LIN {X -0.088,Y -552.932,Z 572.275,A 0.000,B 0.000,C 90.000,E1 265.527} C_DIS
LIN {X -0.264,Y -552.166,Z 572.267,A 0.000,B 0.000,C 90.000,E1 264.147} C_DIS
LIN {X 0.151,Y -551.255,Z 572.260,A 0.000,B 0.000,C 90.000,E1 262.704} C_DIS
LIN {X -0.031,Y -550.259,Z 572.253,A 0.000,B 0.000,C 90.000,E1 261.602} C_DIS
LIN {X -0.102,Y -548.526,Z 572.244,A 0.000,B 0.000,C 90.000,E1 259.926} C_DIS
LIN {X -0.023,Y -546.833,Z 572.235,A 0.000,B 0.000,C 90.000,E1 258.229} C_DIS
LIN {X 0.017,Y -545.061,Z 572.225,A 0.000,B 0.000,C 90.000,E1 256.533} C_DIS
LIN {X 0.274,Y -543.280,Z 572.216,A 0.000,B 0.000,C 90.000,E1 254.810} C_DIS
LIN {X -0.094,Y -541.576,Z 572.208,A 0.000,B 0.000,C 90.000,E1 253.433} C_DIS
LIN {X 0.029,Y -539.678,Z 572.200,A 0.000,B 0.000,C 90.000,E1 252.000} C_DIS
LIN {X 0.055,Y -538.028,Z 572.194,A 0.000,B 0.000,C 90.000,E1 250.859} C_DIS
LIN {X 0.231,Y -536.142,Z 572.187,A 0.000,B 0.000,C 90.000,E1 249.699} C_DIS
LIN {X 0.172,Y -534.661,Z 572.183,A 0.000,B 0.000,C 90.000,E1 248.847} C_DIS
LIN {X 0.198,Y -531.884,Z 572.175,A 0.000,B 0.000,C 90.000,E1 247.411} C_DIS
LIN {X -0.115,Y -528.234,Z 572.165,A 0.000,B 0.000,C 90.000,E1 245.717} C_DIS
LIN {X -0.200,Y -525.022,Z 572.157,A 0.000,B 0.000,C 90.000,E1 244.280} C_DIS
LIN {X 0.109,Y -521.645,Z 572.149,A 0.000,B 0.000,C 90.000,E1 242.794} C_DIS
LIN {X -0.018,Y -518.791,Z 572.143,A 0.000,B 0.000,C 90.000,E1 241.641} C_DIS
LIN {X 0.056,Y -515.801,Z 572.136,A 0.000,B 0.000,C 90.000,E1 240.461} C_DIS
LIN {X 0.080,Y -512.503,Z 572.129,A 0.000,B 0.000,C 90.000,E1 239.282} C_DIS
LIN {X 0.214,Y -508.339,Z 572.121,A 0.000,B 0.000,C 90.000,E1 237.788} C_DIS
LIN {X 0.164,Y -503.280,Z 572.111,A 0.000,B 0.000,C 90.000,E1 236.008} C_DIS
LIN {X -0.001,Y -499.031,Z 572.103,A 0.000,B 0.000,C 90.000,E1 234.529} C_DIS
LIN {X 0.032,Y -492.451,Z 572.090,A 0.000,B 0.000,C 90.000,E1 232.110} C_DIS
LIN {X -0.062,Y -486.845,Z 572.078,A 0.000,B 0.000,C 90.000,E1 229.989} C_DIS
LIN {X -0.046,Y -481.361,Z 572.066,A 0.000,B 0.000,C 90.000,E1 227.838} C_DIS
LIN {X 0.036,Y -476.717,Z 572.055,A 0.000,B 0.000,C 90.000,E1 225.972} C_DIS
LIN {X 0.030,Y -474.441,Z 572.050,A 0.000,B 0.000,C 90.000,E1 225.040} C_DIS
LIN {X 0.182,Y -470.757,Z 572.042,A 0.000,B 0.000,C 90.000,E1 223.461} C_DIS
LIN {X 0.020,Y -466.436,Z 572.031,A 0.000,B 0.000,C 90.000,E1 221.595} C_DIS
LIN {X -0.149,Y -461.582,Z 572.019,A 0.000,B 0.000,C 90.000,E1 219.402} C_DIS
LIN {X -0.024,Y -456.772,Z 572.006,A 0.000,B 0.000,C 90.000,E1 217.156} C_DIS
LIN {X 0.258,Y -453.476,Z 571.998,A 0.000,B 0.000,C 90.000,E1 215.518} C_DIS
LIN {X 0.076,Y -448.240,Z 571.983,A 0.000,B 0.000,C 90.000,E1 212.959} C_DIS
LIN {X 0.188,Y -443.956,Z 571.971,A 0.000,B 0.000,C 90.000,E1 210.669} C_DIS
LIN {X -0.141,Y -440.991,Z 571.961,A 0.000,B 0.000,C 90.000,E1 209.077} C_DIS
LIN {X 0.241,Y -438.187,Z 571.952,A 0.000,B 0.000,C 90.000,E1 207.385} C_DIS
LIN {X -0.204,Y -434.731,Z 571.941,A 0.000,B 0.000,C 90.000,E1 205.463} C_DIS
LIN {X 0.239,Y -432.507,Z 571.934,A 0.000,B 0.000,C 90.000,E1 204.079} C_DIS
LIN {X -0.109,Y -429.841,Z 571.925,A 0.000,B 0.000,C 90.000,E1 202.461} C_DIS
LIN {X -0.108,Y -426.345,Z 571.912,A 0.000,B 0.000,C 90.000,E1 200.120} C_DIS
LIN {X 0.253,Y -423.517,Z 571.901,A 0.000,B 0.000,C 90.000,E1 198.055} C_DIS
LIN {X 0.109,Y -419.981,Z 571.885,A 0.000,B 0.000,C 90.000,E1 195.371} C_DIS
LIN {X -0.104,Y -417.895,Z 571.876,A 0.000,B 0.000,C 90.000,E1 193.703} C_DIS
LIN {X 0.203,Y -415.958,Z 571.869,A 0.000,B 0.000,C 90.000,E1 192.299} C_DIS
LIN {X -0.089,Y -411.389,Z 571.849,A 0.000,B 0.000,C 90.000,E1 188.916} C_DIS
LIN {X 0.052,Y -408.670,Z 571.836,A 0.000,B 0.000,C 90.000,E1 186.486} C_DIS
LIN {X 0.014,Y -406.386,Z 571.825,A 0.000,B 0.000,C 90.000,E1 184.416} C_DIS
LIN {X 0.157,Y -402.836,Z 571.803,A 0.000,B 0.000,C 90.000,E1 180.573} C_DIS
LIN {X -0.095,Y -401.155,Z 571.790,A 0.000,B 0.000,C 90.000,E1 178.165} C_DIS
LIN {X 0.102,Y -400.219,Z 571.780,A 0.000,B 0.000,C 90.000,E1 176.388} C_DIS
LIN {X -0.205,Y -399.268,Z 571.764,A 0.000,B 0.000,C 90.000,E1 173.628} C_DIS
LIN {X 0.011,Y -398.849,Z 571.751,A 0.000,B 0.000,C 90.000,E1 171.141} C_DIS
LIN {X -0.098,Y -398.774,Z 571.739,A 0.000,B 0.000,C 90.000,E1 169.050} C_DIS
LIN {X -0.033,Y -399.127,Z 571.722,A 0.000,B 0.000,C 90.000,E1 165.880} C_DIS
LIN {X -0.088,Y -399.778,Z 571.708,A 0.000,B 0.000,C 90.000,E1 163.433} C_DIS
LIN {X 0.001,Y -400.656,Z 571.694,A 0.000,B 0.000,C 90.000,E1 160.967} C_DIS
LIN {X 0.142,Y -401.621,Z 571.683,A 0.000,B 0.000,C 90.000,E1 158.847} C_DIS
LIN {X -0.157,Y -402.652,Z 571.671,A 0.000,B 0.000,C 90.000,E1 156.794} C_DIS
LIN {X -0.149,Y -403.596,Z 571.661,A 0.000,B 0.000,C 90.000,E1 155.049} C_DIS
LIN {X 0.219,Y -404.546,Z 571.652,A 0.000,B 0.000,C 90.000,E1 153.256} C_DIS
LIN {X -0.108,Y -405.512,Z 571.642,A 0.000,B 0.000,C 90.000,E1 151.563} C_DIS
LIN {X 0.228,Y -406.196,Z 571.634,A 0.000,B 0.000,C 90.000,E1 150.127} C_DIS
LIN {X -0.131,Y -406.783,Z 571.627,A 0.000,B 0.000,C 90.000,E1 148.791} C_DIS
LIN {X -0.008,Y -407.394,Z 571.617,A 0.000,B 0.000,C 90.000,E1 147.041} C_DIS
LIN {X 0.005,Y -407.816,Z 571.607,A 0.000,B 0.000,C 90.000,E1 145.308} C_DIS
LIN {X 0.021,Y -408.164,Z 571.598,A 0.000,B 0.000,C 90.000,E1 143.577} C_DIS
LIN {X 0.198,Y -408.476,Z 571.588,A 0.000,B 0.000,C 90.000,E1 141.823} C_DIS
LIN {X -0.042,Y -408.720,Z 571.577,A 0.000,B 0.000,C 90.000,E1 139.784} C_DIS
LIN {X -0.059,Y -408.883,Z 571.569,A 0.000,B 0.000,C 90.000,E1 138.405} C_DIS
LIN {X 0.199,Y -408.999,Z 571.557,A 0.000,B 0.000,C 90.000,E1 136.296} C_DIS
LIN {X 0.018,Y -409.279,Z 571.544,A 0.000,B 0.000,C 90.000,E1 133.905} C_DIS
LIN {X 0.146,Y -409.500,Z 571.534,A 0.000,B 0.000,C 90.000,E1 132.162} C_DIS
LIN {X 0.148,Y -409.543,Z 571.527,A 0.000,B 0.000,C 90.000,E1 130.782} C_DIS
LIN {X -0.115,Y -409.440,Z 571.519,A 0.000,B 0.000,C 90.000,E1 129.439} C_DIS
LIN {X 0.232,Y -409.205,Z 571.512,A 0.000,B 0.000,C 90.000,E1 128.096} C_DIS
LIN {X 0.098,Y -415.513,Z 571.500,A 0.000,B 0.000,C 90.000,E1 125.964} C_DIS
LIN {X 0.182,Y -425.905,Z 571.477,A 0.000,B 0.000,C 90.000,E1 121.878} C_DIS
LIN {X 0.136,Y -430.920,Z 571.468,A 0.000,B 0.000,C 90.000,E1 120.207} C_DIS
LIN {X 0.004,Y -434.960,Z 571.458,A 0.000,B 0.000,C 90.000,E1 118.487} C_DIS
LIN {X -0.035,Y -434.992,Z 571.458,A 0.000,B 0.000,C 90.000,E1 118.487} C_DIS
LIN {X 0.108,Y -447.698,Z 571.455,A 0.000,B 0.000,C 90.000,E1 117.897} C_DIS
LIN {X -0.098,Y -466.481,Z 571.450,A 0.000,B 0.000,C 90.000,E1 117.052} C_DIS
LIN {X 0.200,Y -474.972,Z 571.448,A 0.000,B 0.000,C 90.000,E1 116.616} C_DIS
LIN {X 0.019,Y -488.662,Z 571.444,A 0.000,B 0.000,C 90.000,E1 115.976} C_DIS
LIN {X 0.304,Y -500.110,Z 571.441,A 0.000,B 0.000,C 90.000,E1 115.335} C_DIS
LIN {X 0.027,Y -511.511,Z 571.437,A 0.000,B 0.000,C 90.000,E1 114.719} C_DIS
LIN {X 0.078,Y -517.954,Z 571.435,A 0.000,B 0.000,C 90.000,E1 114.335} C_DIS
LIN {X -0.215,Y -527.586,Z 571.432,A 0.000,B 0.000,C 90.000,E1 113.770} C_DIS
LIN {X -0.042,Y -536.611,Z 571.429,A 0.000,B 0.000,C 90.000,E1 113.131} C_DIS
LIN {X 0.083,Y -540.758,Z 571.427,A 0.000,B 0.000,C 90.000,E1 112.823} C_DIS
LIN {X 0.012,Y -544.976,Z 571.425,A 0.000,B 0.000,C 90.000,E1 112.514} C_DIS
LIN {X 0.082,Y -550.454,Z 571.423,A 0.000,B 0.000,C 90.000,E1 112.078} C_DIS
LIN {X -0.089,Y -555.613,Z 571.420,A 0.000,B 0.000,C 90.000,E1 111.642} C_DIS
LIN {X 0.113,Y -560.392,Z 571.418,A 0.000,B 0.000,C 90.000,E1 111.173} C_DIS
LIN {X -0.204,Y -564.852,Z 571.415,A 0.000,B 0.000,C 90.000,E1 110.737} C_DIS
LIN {X 0.171,Y -570.133,Z 571.412,A 0.000,B 0.000,C 90.000,E1 110.066} C_DIS
LIN {X 0.048,Y -575.019,Z 571.408,A 0.000,B 0.000,C 90.000,E1 109.396} C_DIS
LIN {X -0.032,Y -579.407,Z 571.404,A 0.000,B 0.000,C 90.000,E1 108.725} C_DIS
LIN {X -0.160,Y -584.107,Z 571.400,A 0.000,B 0.000,C 90.000,E1 107.928} C_DIS
LIN {X 0.211,Y -587.650,Z 571.396,A 0.000,B 0.000,C 90.000,E1 107.221} C_DIS
LIN {X 0.061,Y -591.597,Z 571.391,A 0.000,B 0.000,C 90.000,E1 106.441} C_DIS
LIN {X -0.128,Y -595.301,Z 571.387,A 0.000,B 0.000,C 90.000,E1 105.662} C_DIS
LIN {X 0.290,Y -598.783,Z 571.383,A 0.000,B 0.000,C 90.000,E1 104.828} C_DIS
LIN {X -0.268,Y -603.045,Z 571.377,A 0.000,B 0.000,C 90.000,E1 103.828} C_DIS
LIN {X 0.148,Y -608.165,Z 571.369,A 0.000,B 0.000,C 90.000,E1 102.479} C_DIS
LIN {X -0.287,Y -612.155,Z 571.364,A 0.000,B 0.000,C 90.000,E1 101.478} C_DIS
LIN {X -0.079,Y -616.069,Z 571.358,A 0.000,B 0.000,C 90.000,E1 100.423} C_DIS
LIN {X 0.115,Y -621.760,Z 571.349,A 0.000,B 0.000,C 90.000,E1 98.859} C_DIS
LIN {X -0.188,Y -627.237,Z 571.341,A 0.000,B 0.000,C 90.000,E1 97.352} C_DIS
LIN {X -0.255,Y -631.446,Z 571.334,A 0.000,B 0.000,C 90.000,E1 96.087} C_DIS
LIN {X 0.295,Y -633.757,Z 571.330,A 0.000,B 0.000,C 90.000,E1 95.277} C_DIS
LIN {X -0.086,Y -636.518,Z 571.324,A 0.000,B 0.000,C 90.000,E1 94.302} C_DIS
LIN {X 0.210,Y -638.864,Z 571.318,A 0.000,B 0.000,C 90.000,E1 93.269} C_DIS
LIN {X -0.252,Y -639.970,Z 571.316,A 0.000,B 0.000,C 90.000,E1 92.808} C_DIS
LIN {X 0.301,Y -641.344,Z 571.311,A 0.000,B 0.000,C 90.000,E1 92.007} C_DIS
LIN {X 0.250,Y -642.504,Z 571.307,A 0.000,B 0.000,C 90.000,E1 91.260} C_DIS
LIN {X -0.038,Y -643.700,Z 571.302,A 0.000,B 0.000,C 90.000,E1 90.286} C_DIS
LIN {X -0.082,Y -644.228,Z 571.297,A 0.000,B 0.000,C 90.000,E1 89.542} C_DIS
LIN {X 0.105,Y -644.478,Z 571.295,A 0.000,B 0.000,C 90.000,E1 89.026} C_DIS
LIN {X -0.144,Y -644.538,Z 571.289,A 0.000,B 0.000,C 90.000,E1 88.051} C_DIS
LIN {X -0.184,Y -644.296,Z 571.285,A 0.000,B 0.000,C 90.000,E1 87.306} C_DIS
LIN {X 0.209,Y -643.628,Z 571.279,A 0.000,B 0.000,C 90.000,E1 86.274} C_DIS
LIN {X -0.051,Y -642.536,Z 571.274,A 0.000,B 0.000,C 90.000,E1 85.298} C_DIS
LIN {X -0.025,Y -641.619,Z 571.270,A 0.000,B 0.000,C 90.000,E1 84.546} C_DIS
LIN {X -0.318,Y -640.005,Z 571.264,A 0.000,B 0.000,C 90.000,E1 83.571} C_DIS
LIN {X 0.063,Y -638.030,Z 571.259,A 0.000,B 0.000,C 90.000,E1 82.534} C_DIS
LIN {X 0.058,Y -636.281,Z 571.254,A 0.000,B 0.000,C 90.000,E1 81.781} C_DIS
LIN {X 0.035,Y -634.447,Z 571.250,A 0.000,B 0.000,C 90.000,E1 81.027} C_DIS
LIN {X 0.236,Y -630.960,Z 571.243,A 0.000,B 0.000,C 90.000,E1 79.746} C_DIS
LIN {X -0.240,Y -627.112,Z 571.236,A 0.000,B 0.000,C 90.000,E1 78.522} C_DIS
LIN {X -0.028,Y -625.508,Z 571.233,A 0.000,B 0.000,C 90.000,E1 77.993} C_DIS
LIN {X -0.035,Y -622.884,Z 571.229,A 0.000,B 0.000,C 90.000,E1 77.229} C_DIS
LIN {X 0.148,Y -621.001,Z 571.226,A 0.000,B 0.000,C 90.000,E1 76.700} C_DIS
LIN {X 0.094,Y -617.927,Z 571.222,A 0.000,B 0.000,C 90.000,E1 75.936} C_DIS
LIN {X 0.005,Y -614.677,Z 571.218,A 0.000,B 0.000,C 90.000,E1 75.172} C_DIS
LIN {X -0.163,Y -610.597,Z 571.213,A 0.000,B 0.000,C 90.000,E1 74.283} C_DIS
LIN {X -0.214,Y -606.056,Z 571.208,A 0.000,B 0.000,C 90.000,E1 73.378} C_DIS
LIN {X 0.263,Y -601.137,Z 571.203,A 0.000,B 0.000,C 90.000,E1 72.417} C_DIS
LIN {X 0.212,Y -597.337,Z 571.199,A 0.000,B 0.000,C 90.000,E1 71.764} C_DIS
LIN {X 0.257,Y -592.101,Z 571.194,A 0.000,B 0.000,C 90.000,E1 70.967} C_DIS
LIN {X -0.176,Y -588.386,Z 571.191,A 0.000,B 0.000,C 90.000,E1 70.477} C_DIS
LIN {X -0.145,Y -583.261,Z 571.188,A 0.000,B 0.000,C 90.000,E1 69.806} C_DIS
LIN {X 0.068,Y -577.957,Z 571.184,A 0.000,B 0.000,C 90.000,E1 69.156} C_DIS
LIN {X -0.196,Y -573.030,Z 571.181,A 0.000,B 0.000,C 90.000,E1 68.646} C_DIS
LIN {X 0.178,Y -568.107,Z 571.179,A 0.000,B 0.000,C 90.000,E1 68.103} C_DIS
LIN {X -0.201,Y -563.053,Z 571.176,A 0.000,B 0.000,C 90.000,E1 67.667} C_DIS
LIN {X 0.152,Y -557.756,Z 571.173,A 0.000,B 0.000,C 90.000,E1 67.177} C_DIS
LIN {X -0.122,Y -553.146,Z 571.171,A 0.000,B 0.000,C 90.000,E1 66.847} C_DIS
LIN {X -0.080,Y -546.850,Z 571.169,A 0.000,B 0.000,C 90.000,E1 66.410} C_DIS
LIN {X 0.018,Y -542.062,Z 571.167,A 0.000,B 0.000,C 90.000,E1 66.102} C_DIS
LIN {X 0.139,Y -535.859,Z 571.165,A 0.000,B 0.000,C 90.000,E1 65.741} C_DIS
LIN {X 0.167,Y -527.281,Z 571.163,A 0.000,B 0.000,C 90.000,E1 65.305} C_DIS
LIN {X 0.065,Y -518.444,Z 571.161,A 0.000,B 0.000,C 90.000,E1 64.921} C_DIS
LIN {X -0.272,Y -511.248,Z 571.159,A 0.000,B 0.000,C 90.000,E1 64.665} C_DIS
LIN {X -0.146,Y -488.653,Z 571.154,A 0.000,B 0.000,C 90.000,E1 63.768} C_DIS
LIN {X 0.070,Y -473.164,Z 571.151,A 0.000,B 0.000,C 90.000,E1 63.127} C_DIS
LIN {X 0.116,Y -459.487,Z 571.148,A 0.000,B 0.000,C 90.000,E1 62.538} C_DIS
LIN {X -0.069,Y -456.318,Z 571.147,A 0.000,B 0.000,C 90.000,E1 62.410} C_DIS
LIN {X -0.110,Y -456.279,Z 571.147,A 0.000,B 0.000,C 90.000,E1 62.410} C_DIS
LIN {X 0.276,Y -455.533,Z 571.144,A 0.000,B 0.000,C 90.000,E1 61.897} C_DIS
LIN {X 0.040,Y -445.588,Z 571.119,A 0.000,B 0.000,C 90.000,E1 57.406} C_DIS
LIN {X 0.096,Y -443.812,Z 571.114,A 0.000,B 0.000,C 90.000,E1 56.421} C_DIS
LIN {X -0.115,Y -437.182,Z 571.098,A 0.000,B 0.000,C 90.000,E1 53.703} C_DIS
LIN {X -0.154,Y -437.181,Z 571.098,A 0.000,B 0.000,C 90.000,E1 53.703} C_DIS
LIN {X 0.077,Y -439.358,Z 571.088,A 0.000,B 0.000,C 90.000,E1 51.823} C_DIS
LIN {X 0.260,Y -441.594,Z 571.077,A 0.000,B 0.000,C 90.000,E1 49.828} C_DIS
LIN {X -0.151,Y -443.500,Z 571.068,A 0.000,B 0.000,C 90.000,E1 48.243} C_DIS
LIN {X 0.069,Y -445.310,Z 571.059,A 0.000,B 0.000,C 90.000,E1 46.581} C_DIS
LIN {X 0.013,Y -447.037,Z 571.050,A 0.000,B 0.000,C 90.000,E1 44.960} C_DIS
LIN {X -0.009,Y -448.128,Z 571.043,A 0.000,B 0.000,C 90.000,E1 43.662} C_DIS
LIN {X -0.023,Y -449.052,Z 571.035,A 0.000,B 0.000,C 90.000,E1 42.366} C_DIS
LIN {X 0.001,Y -449.622,Z 571.030,A 0.000,B 0.000,C 90.000,E1 41.391} C_DIS
LIN {X 0.034,Y -450.168,Z 571.023,A 0.000,B 0.000,C 90.000,E1 40.092} C_DIS
LIN {X 0.123,Y -450.506,Z 571.014,A 0.000,B 0.000,C 90.000,E1 38.463} C_DIS
LIN {X 0.176,Y -450.636,Z 571.010,A 0.000,B 0.000,C 90.000,E1 37.810} C_DIS
LIN {X -0.012,Y -450.526,Z 571.001,A 0.000,B 0.000,C 90.000,E1 36.217} C_DIS
LIN {X -0.103,Y -450.233,Z 570.992,A 0.000,B 0.000,C 90.000,E1 34.612} C_DIS
LIN {X -0.044,Y -449.765,Z 570.980,A 0.000,B 0.000,C 90.000,E1 32.339} C_DIS
LIN {X -0.092,Y -449.388,Z 570.967,A 0.000,B 0.000,C 90.000,E1 30.079} C_DIS
LIN {X 0.225,Y -449.212,Z 570.960,A 0.000,B 0.000,C 90.000,E1 28.743} C_DIS
LIN {X 0.179,Y -448.941,Z 570.951,A 0.000,B 0.000,C 90.000,E1 27.129} C_DIS
LIN {X -0.131,Y -448.623,Z 570.938,A 0.000,B 0.000,C 90.000,E1 24.899} C_DIS
LIN {X -0.107,Y -448.456,Z 570.927,A 0.000,B 0.000,C 90.000,E1 22.950} C_DIS
LIN {X -0.021,Y -448.482,Z 570.920,A 0.000,B 0.000,C 90.000,E1 21.642} C_DIS
LIN {X -0.210,Y -448.518,Z 570.908,A 0.000,B 0.000,C 90.000,E1 19.396} C_DIS
LIN {X 0.032,Y -448.730,Z 570.895,A 0.000,B 0.000,C 90.000,E1 17.094} C_DIS
LIN {X 0.008,Y -449.157,Z 570.882,A 0.000,B 0.000,C 90.000,E1 14.828} C_DIS
LIN {X 0.210,Y -449.882,Z 570.870,A 0.000,B 0.000,C 90.000,E1 12.535} C_DIS
LIN {X 0.144,Y -450.729,Z 570.859,A 0.000,B 0.000,C 90.000,E1 10.602} C_DIS
LIN {X 0.143,Y -451.978,Z 570.846,A 0.000,B 0.000,C 90.000,E1 8.341} C_DIS
LIN {X -0.128,Y -453.695,Z 570.832,A 0.000,B 0.000,C 90.000,E1 5.796} C_DIS
LIN {X -0.203,Y -455.559,Z 570.820,A 0.000,B 0.000,C 90.000,E1 3.555} C_DIS
LIN {X 0.012,Y -457.357,Z 570.809,A 0.000,B 0.000,C 90.000,E1 1.604} C_DIS
LIN {X 0.110,Y -460.029,Z 570.795,A 0.000,B 0.000,C 90.000,E1 359.141} C_DIS
LIN {X -0.066,Y -463.334,Z 570.781,A 0.000,B 0.000,C 90.000,E1 356.617} C_DIS
LIN {X -0.122,Y -466.013,Z 570.771,A 0.000,B 0.000,C 90.000,E1 354.723} C_DIS
LIN {X 0.246,Y -469.326,Z 570.758,A 0.000,B 0.000,C 90.000,E1 352.470} C_DIS
LIN {X -0.054,Y -472.137,Z 570.748,A 0.000,B 0.000,C 90.000,E1 350.622} C_DIS
LIN {X 0.155,Y -475.469,Z 570.736,A 0.000,B 0.000,C 90.000,E1 348.409} C_DIS
LIN {X 0.040,Y -479.382,Z 570.722,A 0.000,B 0.000,C 90.000,E1 345.936} C_DIS
LIN {X 0.012,Y -484.890,Z 570.705,A 0.000,B 0.000,C 90.000,E1 342.851} C_DIS
LIN {X -0.239,Y -488.408,Z 570.695,A 0.000,B 0.000,C 90.000,E1 341.040} C_DIS
LIN {X -0.282,Y -491.392,Z 570.686,A 0.000,B 0.000,C 90.000,E1 339.518} C_DIS
LIN {X -0.135,Y -493.688,Z 570.679,A 0.000,B 0.000,C 90.000,E1 338.284} C_DIS
LIN {X 0.100,Y -496.529,Z 570.671,A 0.000,B 0.000,C 90.000,E1 336.741} C_DIS
LIN {X 0.128,Y -499.231,Z 570.663,A 0.000,B 0.000,C 90.000,E1 335.229} C_DIS
LIN {X 0.044,Y -502.287,Z 570.652,A 0.000,B 0.000,C 90.000,E1 333.435} C_DIS
LIN {X -0.043,Y -504.697,Z 570.644,A 0.000,B 0.000,C 90.000,E1 331.948} C_DIS
LIN {X -0.091,Y -507.087,Z 570.636,A 0.000,B 0.000,C 90.000,E1 330.461} C_DIS
LIN {X 0.041,Y -510.039,Z 570.626,A 0.000,B 0.000,C 90.000,E1 328.663} C_DIS
LIN {X 0.141,Y -513.556,Z 570.614,A 0.000,B 0.000,C 90.000,E1 326.580} C_DIS
LIN {X 0.113,Y -516.619,Z 570.605,A 0.000,B 0.000,C 90.000,E1 324.815} C_DIS
LIN {X 0.222,Y -519.230,Z 570.596,A 0.000,B 0.000,C 90.000,E1 323.336} C_DIS
LIN {X 0.141,Y -523.486,Z 570.583,A 0.000,B 0.000,C 90.000,E1 321.009} C_DIS
LIN {X -0.202,Y -527.567,Z 570.572,A 0.000,B 0.000,C 90.000,E1 319.013} C_DIS
LIN {X -0.147,Y -532.109,Z 570.561,A 0.000,B 0.000,C 90.000,E1 316.986} C_DIS
LIN {X -0.308,Y -535.604,Z 570.553,A 0.000,B 0.000,C 90.000,E1 315.567} C_DIS
LIN {X 0.045,Y -536.440,Z 570.551,A 0.000,B 0.000,C 90.000,E1 315.243} C_DIS
LIN {X 0.001,Y -537.927,Z 570.548,A 0.000,B 0.000,C 90.000,E1 314.676} C_DIS
LIN {X -0.031,Y -539.815,Z 570.545,A 0.000,B 0.000,C 90.000,E1 314.109} C_DIS
LIN {X -0.240,Y -541.344,Z 570.543,A 0.000,B 0.000,C 90.000,E1 313.704} C_DIS
LIN {X 0.137,Y -542.937,Z 570.541,A 0.000,B 0.000,C 90.000,E1 313.380} C_DIS
LIN {X -0.045,Y -543.615,Z 570.540,A 0.000,B 0.000,C 90.000,E1 313.257} C_DIS
LIN {X 0.150,Y -544.524,Z 570.540,A 0.000,B 0.000,C 90.000,E1 313.095} C_DIS
LIN {X -0.056,Y -545.632,Z 570.539,A 0.000,B 0.000,C 90.000,E1 312.975} C_DIS
LIN {X -0.036,Y -547.549,Z 570.537,A 0.000,B 0.000,C 90.000,E1 312.690} C_DIS
LIN {X 0.125,Y -550.221,Z 570.535,A 0.000,B 0.000,C 90.000,E1 312.366} C_DIS
LIN {X -0.013,Y -551.276,Z 570.535,A 0.000,B 0.000,C 90.000,E1 312.243} C_DIS
LIN {X 0.208,Y -552.579,Z 570.534,A 0.000,B 0.000,C 90.000,E1 312.081} C_DIS
LIN {X -0.044,Y -560.700,Z 570.530,A 0.000,B 0.000,C 90.000,E1 311.391} C_DIS
LIN {X 0.050,Y -568.069,Z 570.527,A 0.000,B 0.000,C 90.000,E1 310.825} C_DIS
LIN {X -0.065,Y -578.642,Z 570.523,A 0.000,B 0.000,C 90.000,E1 310.092} C_DIS
LIN {X -0.148,Y -593.325,Z 570.517,A 0.000,B 0.000,C 90.000,E1 309.036} C_DIS
LIN {X -0.106,Y -598.899,Z 570.514,A 0.000,B 0.000,C 90.000,E1 308.588} C_DIS
LIN {X 0.204,Y -604.198,Z 570.512,A 0.000,B 0.000,C 90.000,E1 308.096} C_DIS
LIN {X 0.230,Y -611.884,Z 570.508,A 0.000,B 0.000,C 90.000,E1 307.363} C_DIS
LIN {X -0.178,Y -621.354,Z 570.502,A 0.000,B 0.000,C 90.000,E1 306.377} C_DIS
LIN {X -0.035,Y -626.861,Z 570.498,A 0.000,B 0.000,C 90.000,E1 305.724} C_DIS
LIN {X 0.145,Y -634.105,Z 570.494,A 0.000,B 0.000,C 90.000,E1 304.818} C_DIS
LIN {X 0.011,Y -638.081,Z 570.491,A 0.000,B 0.000,C 90.000,E1 304.326} C_DIS
LIN {X -0.058,Y -643.593,Z 570.487,A 0.000,B 0.000,C 90.000,E1 303.579} C_DIS
LIN {X -0.069,Y -648.508,Z 570.482,A 0.000,B 0.000,C 90.000,E1 302.832} C_DIS
LIN {X -0.116,Y -651.476,Z 570.480,A 0.000,B 0.000,C 90.000,E1 302.339} C_DIS
LIN {X 0.112,Y -654.579,Z 570.476,A 0.000,B 0.000,C 90.000,E1 301.720} C_DIS
LIN {X -0.143,Y -658.032,Z 570.472,A 0.000,B 0.000,C 90.000,E1 301.003} C_DIS
LIN {X -0.145,Y -660.216,Z 570.469,A 0.000,B 0.000,C 90.000,E1 300.512} C_DIS
LIN {X 0.232,Y -663.355,Z 570.465,A 0.000,B 0.000,C 90.000,E1 299.745} C_DIS
LIN {X 0.074,Y -666.218,Z 570.461,A 0.000,B 0.000,C 90.000,E1 299.027} C_DIS
LIN {X -0.055,Y -668.888,Z 570.457,A 0.000,B 0.000,C 90.000,E1 298.309} C_DIS
LIN {X -0.161,Y -671.387,Z 570.453,A 0.000,B 0.000,C 90.000,E1 297.590} C_DIS
LIN {X 0.007,Y -672.161,Z 570.452,A 0.000,B 0.000,C 90.000,E1 297.334} C_DIS
LIN {X 0.180,Y -673.103,Z 570.451,A 0.000,B 0.000,C 90.000,E1 297.078} C_DIS
LIN {X 0.110,Y -675.289,Z 570.447,A 0.000,B 0.000,C 90.000,E1 296.360} C_DIS
LIN {X 0.291,Y -675.857,Z 570.445,A 0.000,B 0.000,C 90.000,E1 296.104} C_DIS
LIN {X -0.240,Y -676.015,Z 570.443,A 0.000,B 0.000,C 90.000,E1 295.668} C_DIS
LIN {X -0.053,Y -675.810,Z 570.441,A 0.000,B 0.000,C 90.000,E1 295.412} C_DIS
LIN {X 0.133,Y -674.890,Z 570.440,A 0.000,B 0.000,C 90.000,E1 295.155} C_DIS
LIN {X 0.226,Y -674.324,Z 570.439,A 0.000,B 0.000,C 90.000,E1 295.027} C_DIS
LIN {X -0.204,Y -672.883,Z 570.438,A 0.000,B 0.000,C 90.000,E1 294.823} C_DIS
LIN {X -0.115,Y -671.963,Z 570.437,A 0.000,B 0.000,C 90.000,E1 294.695} C_DIS
LIN {X -0.308,Y -670.456,Z 570.437,A 0.000,B 0.000,C 90.000,E1 294.591} C_DIS
LIN {X -0.126,Y -669.413,Z 570.436,A 0.000,B 0.000,C 90.000,E1 294.515} C_DIS
LIN {X -0.016,Y -666.897,Z 570.435,A 0.000,B 0.000,C 90.000,E1 294.259} C_DIS
LIN {X 0.086,Y -665.372,Z 570.434,A 0.000,B 0.000,C 90.000,E1 294.131} C_DIS
LIN {X 0.061,Y -663.097,Z 570.434,A 0.000,B 0.000,C 90.000,E1 294.027} C_DIS
LIN {X 0.257,Y -657.087,Z 570.432,A 0.000,B 0.000,C 90.000,E1 293.770} C_DIS
LIN {X 0.090,Y -655.093,Z 570.432,A 0.000,B 0.000,C 90.000,E1 293.718} C_DIS
LIN {X -0.292,Y -646.617,Z 570.431,A 0.000,B 0.000,C 90.000,E1 293.515} C_DIS
LIN {X 0.153,Y -628.270,Z 570.428,A 0.000,B 0.000,C 90.000,E1 293.025} C_DIS
LIN {X -0.238,Y -621.422,Z 570.427,A 0.000,B 0.000,C 90.000,E1 292.898} C_DIS
LIN {X 0.179,Y -601.374,Z 570.424,A 0.000,B 0.000,C 90.000,E1 292.280} C_DIS
LIN {X -0.040,Y -580.842,Z 570.420,A 0.000,B 0.000,C 90.000,E1 291.642} C_DIS
LIN {X -0.054,Y -573.123,Z 570.419,A 0.000,B 0.000,C 90.000,E1 291.354} C_DIS
LIN {X -0.135,Y -567.535,Z 570.417,A 0.000,B 0.000,C 90.000,E1 291.099} C_DIS
LIN {X 0.028,Y -564.657,Z 570.416,A 0.000,B 0.000,C 90.000,E1 290.844} C_DIS
LIN {X -0.008,Y -564.624,Z 570.416,A 0.000,B 0.000,C 90.000,E1 290.844} C_DIS
LIN {X -0.016,Y -563.935,Z 570.415,A 0.000,B 0.000,C 90.000,E1 290.663} C_DIS
LIN {X 0.055,Y -563.651,Z 570.412,A 0.000,B 0.000,C 90.000,E1 290.174} C_DIS
LIN {X -0.099,Y -563.715,Z 570.406,A 0.000,B 0.000,C 90.000,E1 289.087} C_DIS
LIN {X -0.250,Y -563.588,Z 570.400,A 0.000,B 0.000,C 90.000,E1 288.000} C_DIS
LIN {X 0.134,Y -563.220,Z 570.394,A 0.000,B 0.000,C 90.000,E1 286.858} C_DIS
LIN {X 0.114,Y -562.582,Z 570.386,A 0.000,B 0.000,C 90.000,E1 285.481} C_DIS
LIN {X -0.071,Y -561.825,Z 570.378,A 0.000,B 0.000,C 90.000,E1 284.120} C_DIS
LIN {X -0.091,Y -560.706,Z 570.368,A 0.000,B 0.000,C 90.000,E1 282.187} C_DIS
LIN {X 0.118,Y -559.882,Z 570.360,A 0.000,B 0.000,C 90.000,E1 280.782} C_DIS
LIN {X -0.197,Y -558.918,Z 570.351,A 0.000,B 0.000,C 90.000,E1 279.151} C_DIS
LIN {X 0.203,Y -557.912,Z 570.338,A 0.000,B 0.000,C 90.000,E1 276.891} C_DIS
LIN {X 0.113,Y -557.375,Z 570.331,A 0.000,B 0.000,C 90.000,E1 275.511} C_DIS
LIN {X 0.136,Y -556.748,Z 570.321,A 0.000,B 0.000,C 90.000,E1 273.841} C_DIS
LIN {X 0.070,Y -556.230,Z 570.312,A 0.000,B 0.000,C 90.000,E1 272.178} C_DIS
LIN {X -0.080,Y -555.687,Z 570.304,A 0.000,B 0.000,C 90.000,E1 270.802} C_DIS
LIN {X 0.226,Y -555.222,Z 570.298,A 0.000,B 0.000,C 90.000,E1 269.656} C_DIS
LIN {X 0.131,Y -554.528,Z 570.289,A 0.000,B 0.000,C 90.000,E1 267.993} C_DIS
LIN {X -0.046,Y -553.898,Z 570.281,A 0.000,B 0.000,C 90.000,E1 266.617} C_DIS
LIN {X -0.140,Y -552.995,Z 570.272,A 0.000,B 0.000,C 90.000,E1 264.951} C_DIS
LIN {X 0.232,Y -552.180,Z 570.264,A 0.000,B 0.000,C 90.000,E1 263.514} C_DIS
LIN {X 0.058,Y -551.369,Z 570.258,A 0.000,B 0.000,C 90.000,E1 262.413} C_DIS
LIN {X -0.118,Y -550.350,Z 570.252,A 0.000,B 0.000,C 90.000,E1 261.310} C_DIS
LIN {X -0.186,Y -548.574,Z 570.242,A 0.000,B 0.000,C 90.000,E1 259.634} C_DIS
LIN {X -0.205,Y -547.174,Z 570.235,A 0.000,B 0.000,C 90.000,E1 258.229} C_DIS
LIN {X -0.029,Y -545.397,Z 570.225,A 0.000,B 0.000,C 90.000,E1 256.520} C_DIS
LIN {X 0.108,Y -543.583,Z 570.216,A 0.000,B 0.000,C 90.000,E1 254.810} C_DIS
LIN {X 0.266,Y -541.844,Z 570.208,A 0.000,B 0.000,C 90.000,E1 253.378} C_DIS
LIN {X -0.128,Y -539.912,Z 570.200,A 0.000,B 0.000,C 90.000,E1 252.000} C_DIS
LIN {X -0.097,Y -538.209,Z 570.194,A 0.000,B 0.000,C 90.000,E1 250.859} C_DIS
LIN {X -0.206,Y -535.813,Z 570.186,A 0.000,B 0.000,C 90.000,E1 249.444} C_DIS
LIN {X -0.265,Y -534.236,Z 570.181,A 0.000,B 0.000,C 90.000,E1 248.592} C_DIS
LIN {X 0.055,Y -532.011,Z 570.175,A 0.000,B 0.000,C 90.000,E1 247.411} C_DIS
LIN {X 0.227,Y -528.355,Z 570.165,A 0.000,B 0.000,C 90.000,E1 245.665} C_DIS
LIN {X 0.136,Y -525.115,Z 570.157,A 0.000,B 0.000,C 90.000,E1 244.229} C_DIS
LIN {X -0.025,Y -521.695,Z 570.149,A 0.000,B 0.000,C 90.000,E1 242.794} C_DIS
LIN {X -0.151,Y -518.826,Z 570.142,A 0.000,B 0.000,C 90.000,E1 241.641} C_DIS
LIN {X -0.077,Y -515.831,Z 570.136,A 0.000,B 0.000,C 90.000,E1 240.461} C_DIS
LIN {X -0.051,Y -512.531,Z 570.129,A 0.000,B 0.000,C 90.000,E1 239.282} C_DIS
LIN {X -0.012,Y -507.402,Z 570.120,A 0.000,B 0.000,C 90.000,E1 237.502} C_DIS
LIN {X 0.035,Y -503.184,Z 570.111,A 0.000,B 0.000,C 90.000,E1 236.008} C_DIS
LIN {X 0.276,Y -498.935,Z 570.103,A 0.000,B 0.000,C 90.000,E1 234.482} C_DIS
LIN {X -0.099,Y -492.378,Z 570.089,A 0.000,B 0.000,C 90.000,E1 232.110} C_DIS
LIN {X -0.193,Y -486.767,Z 570.078,A 0.000,B 0.000,C 90.000,E1 229.989} C_DIS
LIN {X 0.178,Y -481.295,Z 570.066,A 0.000,B 0.000,C 90.000,E1 227.796} C_DIS
LIN {X 0.126,Y -475.144,Z 570.052,A 0.000,B 0.000,C 90.000,E1 225.324} C_DIS
LIN {X 0.048,Y -470.689,Z 570.042,A 0.000,B 0.000,C 90.000,E1 223.461} C_DIS
LIN {X -0.184,Y -467.086,Z 570.033,A 0.000,B 0.000,C 90.000,E1 221.919} C_DIS
LIN {X -0.032,Y -462.151,Z 570.021,A 0.000,B 0.000,C 90.000,E1 219.688} C_DIS
LIN {X 0.244,Y -459.399,Z 570.013,A 0.000,B 0.000,C 90.000,E1 218.382} C_DIS
LIN {X -0.058,Y -455.325,Z 570.003,A 0.000,B 0.000,C 90.000,E1 216.503} C_DIS
LIN {X -0.157,Y -452.660,Z 569.996,A 0.000,B 0.000,C 90.000,E1 215.231} C_DIS
LIN {X -0.063,Y -448.112,Z 569.983,A 0.000,B 0.000,C 90.000,E1 212.959} C_DIS
LIN {X -0.017,Y -444.404,Z 569.972,A 0.000,B 0.000,C 90.000,E1 211.003} C_DIS
LIN {X 0.050,Y -441.451,Z 569.963,A 0.000,B 0.000,C 90.000,E1 209.361} C_DIS
LIN {X 0.095,Y -438.024,Z 569.952,A 0.000,B 0.000,C 90.000,E1 207.385} C_DIS
LIN {X 0.215,Y -435.164,Z 569.943,A 0.000,B 0.000,C 90.000,E1 205.720} C_DIS
LIN {X -0.101,Y -431.317,Z 569.930,A 0.000,B 0.000,C 90.000,E1 203.439} C_DIS
LIN {X -0.063,Y -426.718,Z 569.914,A 0.000,B 0.000,C 90.000,E1 200.429} C_DIS
LIN {X 0.120,Y -424.344,Z 569.904,A 0.000,B 0.000,C 90.000,E1 198.725} C_DIS
LIN {X -0.105,Y -421.587,Z 569.893,A 0.000,B 0.000,C 90.000,E1 196.732} C_DIS
LIN {X -0.229,Y -419.078,Z 569.882,A 0.000,B 0.000,C 90.000,E1 194.717} C_DIS
LIN {X 0.143,Y -417.823,Z 569.876,A 0.000,B 0.000,C 90.000,E1 193.647} C_DIS
LIN {X -0.007,Y -416.400,Z 569.870,A 0.000,B 0.000,C 90.000,E1 192.647} C_DIS
LIN {X 0.085,Y -412.186,Z 569.853,A 0.000,B 0.000,C 90.000,E1 189.557} C_DIS
LIN {X -0.106,Y -408.671,Z 569.836,A 0.000,B 0.000,C 90.000,E1 186.486} C_DIS
LIN {X -0.143,Y -406.412,Z 569.824,A 0.000,B 0.000,C 90.000,E1 184.416} C_DIS
LIN {X 0.003,Y -402.913,Z 569.803,A 0.000,B 0.000,C 90.000,E1 180.573} C_DIS
LIN {X 0.184,Y -401.471,Z 569.792,A 0.000,B 0.000,C 90.000,E1 178.453} C_DIS
LIN {X 0.000,Y -400.500,Z 569.782,A 0.000,B 0.000,C 90.000,E1 176.731} C_DIS
LIN {X 0.107,Y -399.470,Z 569.766,A 0.000,B 0.000,C 90.000,E1 173.913} C_DIS
LIN {X -0.132,Y -398.970,Z 569.751,A 0.000,B 0.000,C 90.000,E1 171.141} C_DIS
LIN {X 0.154,Y -398.895,Z 569.739,A 0.000,B 0.000,C 90.000,E1 168.993} C_DIS
LIN {X -0.168,Y -399.254,Z 569.721,A 0.000,B 0.000,C 90.000,E1 165.880} C_DIS
LIN {X 0.003,Y -399.711,Z 569.712,A 0.000,B 0.000,C 90.000,E1 164.102} C_DIS
LIN {X 0.165,Y -400.674,Z 569.696,A 0.000,B 0.000,C 90.000,E1 161.275} C_DIS
LIN {X -0.069,Y -401.620,Z 569.685,A 0.000,B 0.000,C 90.000,E1 159.209} C_DIS
LIN {X 0.006,Y -402.629,Z 569.673,A 0.000,B 0.000,C 90.000,E1 157.102} C_DIS
LIN {X 0.017,Y -403.595,Z 569.663,A 0.000,B 0.000,C 90.000,E1 155.357} C_DIS
LIN {X 0.104,Y -404.739,Z 569.652,A 0.000,B 0.000,C 90.000,E1 153.256} C_DIS
LIN {X 0.138,Y -405.720,Z 569.642,A 0.000,B 0.000,C 90.000,E1 151.513} C_DIS
LIN {X 0.120,Y -406.402,Z 569.634,A 0.000,B 0.000,C 90.000,E1 150.127} C_DIS
LIN {X 0.113,Y -407.008,Z 569.626,A 0.000,B 0.000,C 90.000,E1 148.742} C_DIS
LIN {X -0.109,Y -407.637,Z 569.617,A 0.000,B 0.000,C 90.000,E1 147.041} C_DIS
LIN {X -0.090,Y -408.057,Z 569.607,A 0.000,B 0.000,C 90.000,E1 145.308} C_DIS
LIN {X -0.070,Y -408.396,Z 569.598,A 0.000,B 0.000,C 90.000,E1 143.577} C_DIS
LIN {X 0.111,Y -408.698,Z 569.588,A 0.000,B 0.000,C 90.000,E1 141.823} C_DIS
LIN {X 0.149,Y -408.872,Z 569.580,A 0.000,B 0.000,C 90.000,E1 140.436} C_DIS
LIN {X -0.135,Y -409.069,Z 569.569,A 0.000,B 0.000,C 90.000,E1 138.405} C_DIS
LIN {X 0.127,Y -409.184,Z 569.557,A 0.000,B 0.000,C 90.000,E1 136.296} C_DIS
LIN {X 0.234,Y -409.462,Z 569.544,A 0.000,B 0.000,C 90.000,E1 133.866} C_DIS
LIN {X 0.082,Y -409.681,Z 569.534,A 0.000,B 0.000,C 90.000,E1 132.162} C_DIS
LIN {X 0.088,Y -409.724,Z 569.527,A 0.000,B 0.000,C 90.000,E1 130.782} C_DIS
LIN {X 0.087,Y -409.611,Z 569.519,A 0.000,B 0.000,C 90.000,E1 129.402} C_DIS
LIN {X -0.131,Y -409.346,Z 569.512,A 0.000,B 0.000,C 90.000,E1 128.096} C_DIS
LIN {X 0.043,Y -415.536,Z 569.500,A 0.000,B 0.000,C 90.000,E1 125.964} C_DIS
LIN {X 0.126,Y -425.926,Z 569.477,A 0.000,B 0.000,C 90.000,E1 121.878} C_DIS
LIN {X 0.080,Y -430.937,Z 569.468,A 0.000,B 0.000,C 90.000,E1 120.207} C_DIS
LIN {X -0.075,Y -435.623,Z 569.457,A 0.000,B 0.000,C 90.000,E1 118.231} C_DIS
LIN {X -0.112,Y -435.698,Z 569.457,A 0.000,B 0.000,C 90.000,E1 118.231} C_DIS
LIN {X -0.058,Y -442.880,Z 569.455,A 0.000,B 0.000,C 90.000,E1 117.897} C_DIS
LIN {X 0.248,Y -461.609,Z 569.450,A 0.000,B 0.000,C 90.000,E1 117.001} C_DIS
LIN {X 0.141,Y -470.241,Z 569.448,A 0.000,B 0.000,C 90.000,E1 116.616} C_DIS
LIN {X -0.246,Y -487.281,Z 569.443,A 0.000,B 0.000,C 90.000,E1 115.848} C_DIS
LIN {X 0.123,Y -498.819,Z 569.440,A 0.000,B 0.000,C 90.000,E1 115.207} C_DIS
LIN {X -0.066,Y -510.279,Z 569.437,A 0.000,B 0.000,C 90.000,E1 114.591} C_DIS
LIN {X 0.046,Y -516.743,Z 569.435,A 0.000,B 0.000,C 90.000,E1 114.207} C_DIS
LIN {X -0.150,Y -526.423,Z 569.431,A 0.000,B 0.000,C 90.000,E1 113.643} C_DIS
LIN {X 0.189,Y -537.119,Z 569.427,A 0.000,B 0.000,C 90.000,E1 112.898} C_DIS
LIN {X -0.065,Y -544.456,Z 569.424,A 0.000,B 0.000,C 90.000,E1 112.386} C_DIS
LIN {X 0.142,Y -549.034,Z 569.422,A 0.000,B 0.000,C 90.000,E1 112.025} C_DIS
LIN {X -0.032,Y -554.402,Z 569.420,A 0.000,B 0.000,C 90.000,E1 111.589} C_DIS
LIN {X 0.297,Y -559.475,Z 569.417,A 0.000,B 0.000,C 90.000,E1 111.099} C_DIS
LIN {X -0.029,Y -564.615,Z 569.415,A 0.000,B 0.000,C 90.000,E1 110.610} C_DIS
LIN {X -0.031,Y -569.267,Z 569.411,A 0.000,B 0.000,C 90.000,E1 110.066} C_DIS
LIN {X -0.161,Y -574.379,Z 569.408,A 0.000,B 0.000,C 90.000,E1 109.396} C_DIS
LIN {X 0.214,Y -579.703,Z 569.403,A 0.000,B 0.000,C 90.000,E1 108.544} C_DIS
LIN {X 0.171,Y -583.728,Z 569.399,A 0.000,B 0.000,C 90.000,E1 107.873} C_DIS
LIN {X -0.094,Y -588.065,Z 569.395,A 0.000,B 0.000,C 90.000,E1 107.094} C_DIS
LIN {X -0.245,Y -591.499,Z 569.391,A 0.000,B 0.000,C 90.000,E1 106.441} C_DIS
LIN {X 0.138,Y -595.322,Z 569.387,A 0.000,B 0.000,C 90.000,E1 105.607} C_DIS
LIN {X -0.016,Y -598.897,Z 569.382,A 0.000,B 0.000,C 90.000,E1 104.828} C_DIS
LIN {X 0.050,Y -605.410,Z 569.374,A 0.000,B 0.000,C 90.000,E1 103.244} C_DIS
LIN {X -0.080,Y -610.590,Z 569.366,A 0.000,B 0.000,C 90.000,E1 101.951} C_DIS
LIN {X -0.134,Y -615.559,Z 569.359,A 0.000,B 0.000,C 90.000,E1 100.658} C_DIS
LIN {X -0.179,Y -622.243,Z 569.349,A 0.000,B 0.000,C 90.000,E1 98.859} C_DIS
LIN {X -0.252,Y -626.844,Z 569.342,A 0.000,B 0.000,C 90.000,E1 97.587} C_DIS
LIN {X 0.256,Y -629.524,Z 569.338,A 0.000,B 0.000,C 90.000,E1 96.777} C_DIS
LIN {X -0.120,Y -632.849,Z 569.332,A 0.000,B 0.000,C 90.000,E1 95.796} C_DIS
LIN {X -0.248,Y -635.095,Z 569.328,A 0.000,B 0.000,C 90.000,E1 95.049} C_DIS
LIN {X 0.071,Y -637.791,Z 569.322,A 0.000,B 0.000,C 90.000,E1 94.012} C_DIS
LIN {X -0.260,Y -640.175,Z 569.317,A 0.000,B 0.000,C 90.000,E1 93.037} C_DIS
LIN {X 0.292,Y -641.626,Z 569.313,A 0.000,B 0.000,C 90.000,E1 92.236} C_DIS
LIN {X 0.244,Y -642.847,Z 569.308,A 0.000,B 0.000,C 90.000,E1 91.489} C_DIS
LIN {X 0.189,Y -643.843,Z 569.304,A 0.000,B 0.000,C 90.000,E1 90.745} C_DIS
LIN {X 0.146,Y -644.659,Z 569.300,A 0.000,B 0.000,C 90.000,E1 90.000} C_DIS
LIN {X -0.116,Y -645.176,Z 569.295,A 0.000,B 0.000,C 90.000,E1 89.026} C_DIS
LIN {X 0.289,Y -645.210,Z 569.289,A 0.000,B 0.000,C 90.000,E1 87.993} C_DIS
LIN {X 0.254,Y -644.952,Z 569.285,A 0.000,B 0.000,C 90.000,E1 87.249} C_DIS
LIN {X 0.014,Y -644.255,Z 569.279,A 0.000,B 0.000,C 90.000,E1 86.274} C_DIS
LIN {X -0.239,Y -643.124,Z 569.274,A 0.000,B 0.000,C 90.000,E1 85.298} C_DIS
LIN {X -0.206,Y -642.196,Z 569.270,A 0.000,B 0.000,C 90.000,E1 84.546} C_DIS
LIN {X 0.145,Y -640.522,Z 569.264,A 0.000,B 0.000,C 90.000,E1 83.514} C_DIS
LIN {X -0.103,Y -638.479,Z 569.259,A 0.000,B 0.000,C 90.000,E1 82.534} C_DIS
LIN {X -0.104,Y -636.723,Z 569.254,A 0.000,B 0.000,C 90.000,E1 81.781} C_DIS
LIN {X -0.120,Y -634.827,Z 569.250,A 0.000,B 0.000,C 90.000,E1 81.027} C_DIS
LIN {X 0.087,Y -631.268,Z 569.243,A 0.000,B 0.000,C 90.000,E1 79.746} C_DIS
LIN {X 0.232,Y -627.357,Z 569.236,A 0.000,B 0.000,C 90.000,E1 78.465} C_DIS
LIN {X -0.170,Y -625.719,Z 569.233,A 0.000,B 0.000,C 90.000,E1 77.993} C_DIS
LIN {X -0.174,Y -623.016,Z 569.229,A 0.000,B 0.000,C 90.000,E1 77.229} C_DIS
LIN {X 0.011,Y -621.091,Z 569.226,A 0.000,B 0.000,C 90.000,E1 76.700} C_DIS
LIN {X -0.042,Y -617.911,Z 569.222,A 0.000,B 0.000,C 90.000,E1 75.936} C_DIS
LIN {X -0.130,Y -614.565,Z 569.218,A 0.000,B 0.000,C 90.000,E1 75.172} C_DIS
LIN {X -0.094,Y -610.999,Z 569.213,A 0.000,B 0.000,C 90.000,E1 74.393} C_DIS
LIN {X -0.307,Y -606.381,Z 569.208,A 0.000,B 0.000,C 90.000,E1 73.504} C_DIS
LIN {X 0.171,Y -601.393,Z 569.203,A 0.000,B 0.000,C 90.000,E1 72.543} C_DIS
LIN {X 0.068,Y -596.649,Z 569.199,A 0.000,B 0.000,C 90.000,E1 71.764} C_DIS
LIN {X -0.180,Y -592.365,Z 569.195,A 0.000,B 0.000,C 90.000,E1 71.148} C_DIS
LIN {X -0.113,Y -587.581,Z 569.192,A 0.000,B 0.000,C 90.000,E1 70.477} C_DIS
LIN {X -0.090,Y -582.243,Z 569.188,A 0.000,B 0.000,C 90.000,E1 69.806} C_DIS
LIN {X -0.038,Y -577.612,Z 569.185,A 0.000,B 0.000,C 90.000,E1 69.263} C_DIS
LIN {X -0.006,Y -571.259,Z 569.181,A 0.000,B 0.000,C 90.000,E1 68.592} C_DIS
LIN {X -0.089,Y -567.335,Z 569.179,A 0.000,B 0.000,C 90.000,E1 68.209} C_DIS
LIN {X -0.254,Y -563.230,Z 569.177,A 0.000,B 0.000,C 90.000,E1 67.847} C_DIS
LIN {X -0.110,Y -557.511,Z 569.174,A 0.000,B 0.000,C 90.000,E1 67.358} C_DIS
LIN {X 0.138,Y -552.763,Z 569.172,A 0.000,B 0.000,C 90.000,E1 66.975} C_DIS
LIN {X 0.230,Y -546.382,Z 569.170,A 0.000,B 0.000,C 90.000,E1 66.538} C_DIS
LIN {X 0.052,Y -540.013,Z 569.168,A 0.000,B 0.000,C 90.000,E1 66.177} C_DIS
LIN {X -0.088,Y -533.449,Z 569.166,A 0.000,B 0.000,C 90.000,E1 65.845} C_DIS
LIN {X 0.141,Y -526.642,Z 569.164,A 0.000,B 0.000,C 90.000,E1 65.485} C_DIS
LIN {X -0.025,Y -516.116,Z 569.161,A 0.000,B 0.000,C 90.000,E1 65.049} C_DIS
LIN {X -0.284,Y -508.961,Z 569.160,A 0.000,B 0.000,C 90.000,E1 64.793} C_DIS
LIN {X -0.065,Y -486.236,Z 569.155,A 0.000,B 0.000,C 90.000,E1 63.896} C_DIS
LIN {X -0.072,Y -465.751,Z 569.150,A 0.000,B 0.000,C 90.000,E1 63.076} C_DIS
LIN {X 0.006,Y -456.823,Z 569.148,A 0.000,B 0.000,C 90.000,E1 62.666} C_DIS
LIN {X -0.033,Y -456.723,Z 569.148,A 0.000,B 0.000,C 90.000,E1 62.666} C_DIS
LIN {X 0.060,Y -455.612,Z 569.144,A 0.000,B 0.000,C 90.000,E1 61.975} C_DIS
LIN {X 0.147,Y -453.304,Z 569.139,A 0.000,B 0.000,C 90.000,E1 61.001} C_DIS
LIN {X -0.183,Y -444.503,Z 569.116,A 0.000,B 0.000,C 90.000,E1 56.834} C_DIS
LIN {X -0.122,Y -443.928,Z 569.114,A 0.000,B 0.000,C 90.000,E1 56.501} C_DIS
LIN {X 0.001,Y -437.569,Z 569.099,A 0.000,B 0.000,C 90.000,E1 53.863} C_DIS
LIN {X -0.038,Y -437.563,Z 569.099,A 0.000,B 0.000,C 90.000,E1 53.863} C_DIS
LIN {X -0.133,Y -439.942,Z 569.088,A 0.000,B 0.000,C 90.000,E1 51.904} C_DIS
LIN {X 0.101,Y -441.872,Z 569.079,A 0.000,B 0.000,C 90.000,E1 50.231} C_DIS
LIN {X -0.018,Y -443.836,Z 569.070,A 0.000,B 0.000,C 90.000,E1 48.609} C_DIS
LIN {X -0.106,Y -446.082,Z 569.059,A 0.000,B 0.000,C 90.000,E1 46.662} C_DIS
LIN {X 0.169,Y -447.821,Z 569.050,A 0.000,B 0.000,C 90.000,E1 45.000} C_DIS
LIN {X 0.156,Y -448.692,Z 569.045,A 0.000,B 0.000,C 90.000,E1 44.028} C_DIS
LIN {X -0.158,Y -449.642,Z 569.038,A 0.000,B 0.000,C 90.000,E1 42.771} C_DIS
LIN {X 0.175,Y -450.263,Z 569.032,A 0.000,B 0.000,C 90.000,E1 41.757} C_DIS
LIN {X 0.215,Y -450.833,Z 569.025,A 0.000,B 0.000,C 90.000,E1 40.458} C_DIS
LIN {X -0.024,Y -451.096,Z 569.020,A 0.000,B 0.000,C 90.000,E1 39.519} C_DIS
LIN {X 0.087,Y -451.363,Z 569.011,A 0.000,B 0.000,C 90.000,E1 37.890} C_DIS
LIN {X -0.083,Y -451.233,Z 569.002,A 0.000,B 0.000,C 90.000,E1 36.297} C_DIS
LIN {X 0.129,Y -450.999,Z 568.994,A 0.000,B 0.000,C 90.000,E1 34.978} C_DIS
LIN {X -0.160,Y -450.443,Z 568.982,A 0.000,B 0.000,C 90.000,E1 32.752} C_DIS
LIN {X 0.042,Y -450.028,Z 568.969,A 0.000,B 0.000,C 90.000,E1 30.463} C_DIS
LIN {X 0.148,Y -449.829,Z 568.962,A 0.000,B 0.000,C 90.000,E1 29.155} C_DIS
LIN {X -0.069,Y -449.539,Z 568.953,A 0.000,B 0.000,C 90.000,E1 27.564} C_DIS
LIN {X 0.034,Y -449.156,Z 568.941,A 0.000,B 0.000,C 90.000,E1 25.283} C_DIS
LIN {X -0.048,Y -448.892,Z 568.928,A 0.000,B 0.000,C 90.000,E1 23.025} C_DIS
LIN {X -0.071,Y -448.878,Z 568.919,A 0.000,B 0.000,C 90.000,E1 21.408} C_DIS
LIN {X 0.033,Y -448.863,Z 568.908,A 0.000,B 0.000,C 90.000,E1 19.450} C_DIS
LIN {X 0.147,Y -449.048,Z 568.896,A 0.000,B 0.000,C 90.000,E1 17.166} C_DIS
LIN {X 0.143,Y -449.431,Z 568.883,A 0.000,B 0.000,C 90.000,E1 14.898} C_DIS
LIN {X -0.018,Y -449.908,Z 568.874,A 0.000,B 0.000,C 90.000,E1 13.300} C_DIS
LIN {X -0.041,Y -450.934,Z 568.860,A 0.000,B 0.000,C 90.000,E1 10.715} C_DIS
LIN {X 0.159,Y -452.343,Z 568.845,A 0.000,B 0.000,C 90.000,E1 8.106} C_DIS
LIN {X 0.049,Y -454.331,Z 568.829,A 0.000,B 0.000,C 90.000,E1 5.220} C_DIS
LIN {X -0.012,Y -456.216,Z 568.817,A 0.000,B 0.000,C 90.000,E1 2.980} C_DIS
LIN {X -0.068,Y -458.387,Z 568.804,A 0.000,B 0.000,C 90.000,E1 0.745} C_DIS
LIN {X -0.209,Y -461.320,Z 568.790,A 0.000,B 0.000,C 90.000,E1 358.224} C_DIS
LIN {X -0.062,Y -463.459,Z 568.781,A 0.000,B 0.000,C 90.000,E1 356.617} C_DIS
LIN {X 0.144,Y -466.566,Z 568.769,A 0.000,B 0.000,C 90.000,E1 354.375} C_DIS
LIN {X 0.257,Y -469.420,Z 568.758,A 0.000,B 0.000,C 90.000,E1 352.470} C_DIS
LIN {X 0.211,Y -471.726,Z 568.750,A 0.000,B 0.000,C 90.000,E1 350.905} C_DIS
LIN {X -0.131,Y -475.036,Z 568.737,A 0.000,B 0.000,C 90.000,E1 348.757} C_DIS
LIN {X 0.096,Y -477.401,Z 568.729,A 0.000,B 0.000,C 90.000,E1 347.173} C_DIS
LIN {X -0.126,Y -480.447,Z 568.719,A 0.000,B 0.000,C 90.000,E1 345.338} C_DIS
LIN {X 0.031,Y -485.533,Z 568.703,A 0.000,B 0.000,C 90.000,E1 342.543} C_DIS
LIN {X -0.201,Y -489.059,Z 568.693,A 0.000,B 0.000,C 90.000,E1 340.732} C_DIS
LIN {X -0.228,Y -492.030,Z 568.684,A 0.000,B 0.000,C 90.000,E1 339.209} C_DIS
LIN {X -0.069,Y -494.265,Z 568.678,A 0.000,B 0.000,C 90.000,E1 337.975} C_DIS
LIN {X 0.174,Y -497.137,Z 568.669,A 0.000,B 0.000,C 90.000,E1 336.433} C_DIS
LIN {X -0.241,Y -499.825,Z 568.661,A 0.000,B 0.000,C 90.000,E1 334.973} C_DIS
LIN {X 0.137,Y -502.870,Z 568.651,A 0.000,B 0.000,C 90.000,E1 333.127} C_DIS
LIN {X 0.055,Y -505.263,Z 568.643,A 0.000,B 0.000,C 90.000,E1 331.641} C_DIS
LIN {X -0.062,Y -507.207,Z 568.636,A 0.000,B 0.000,C 90.000,E1 330.461} C_DIS
LIN {X -0.029,Y -510.654,Z 568.624,A 0.000,B 0.000,C 90.000,E1 328.377} C_DIS
LIN {X 0.094,Y -514.189,Z 568.613,A 0.000,B 0.000,C 90.000,E1 326.294} C_DIS
LIN {X 0.153,Y -516.765,Z 568.605,A 0.000,B 0.000,C 90.000,E1 324.815} C_DIS
LIN {X 0.263,Y -519.371,Z 568.596,A 0.000,B 0.000,C 90.000,E1 323.336} C_DIS
LIN {X 0.186,Y -523.618,Z 568.584,A 0.000,B 0.000,C 90.000,E1 321.009} C_DIS
LIN {X -0.152,Y -527.717,Z 568.572,A 0.000,B 0.000,C 90.000,E1 319.013} C_DIS
LIN {X 0.324,Y -531.574,Z 568.563,A 0.000,B 0.000,C 90.000,E1 317.229} C_DIS
LIN {X 0.037,Y -538.642,Z 568.547,A 0.000,B 0.000,C 90.000,E1 314.393} C_DIS
LIN {X -0.348,Y -540.565,Z 568.544,A 0.000,B 0.000,C 90.000,E1 313.866} C_DIS
LIN {X 0.024,Y -541.405,Z 568.542,A 0.000,B 0.000,C 90.000,E1 313.542} C_DIS
LIN {X 0.029,Y -542.433,Z 568.540,A 0.000,B 0.000,C 90.000,E1 313.257} C_DIS
LIN {X 0.012,Y -543.845,Z 568.539,A 0.000,B 0.000,C 90.000,E1 312.975} C_DIS
LIN {X 0.119,Y -545.997,Z 568.537,A 0.000,B 0.000,C 90.000,E1 312.609} C_DIS
LIN {X -0.034,Y -551.441,Z 568.533,A 0.000,B 0.000,C 90.000,E1 311.919} C_DIS
LIN {X 0.094,Y -555.851,Z 568.531,A 0.000,B 0.000,C 90.000,E1 311.472} C_DIS
LIN {X -0.012,Y -561.193,Z 568.528,A 0.000,B 0.000,C 90.000,E1 311.024} C_DIS
LIN {X -0.114,Y -569.835,Z 568.524,A 0.000,B 0.000,C 90.000,E1 310.378} C_DIS
LIN {X -0.140,Y -577.457,Z 568.521,A 0.000,B 0.000,C 90.000,E1 309.850} C_DIS
LIN {X 0.200,Y -592.164,Z 568.515,A 0.000,B 0.000,C 90.000,E1 308.749} C_DIS
LIN {X -0.100,Y -597.656,Z 568.513,A 0.000,B 0.000,C 90.000,E1 308.338} C_DIS
LIN {X -0.271,Y -603.006,Z 568.510,A 0.000,B 0.000,C 90.000,E1 307.890} C_DIS
LIN {X -0.285,Y -610.705,Z 568.506,A 0.000,B 0.000,C 90.000,E1 307.156} C_DIS
LIN {X -0.038,Y -616.678,Z 568.503,A 0.000,B 0.000,C 90.000,E1 306.503} C_DIS
LIN {X 0.264,Y -620.191,Z 568.501,A 0.000,B 0.000,C 90.000,E1 306.091} C_DIS
LIN {X 0.118,Y -625.601,Z 568.497,A 0.000,B 0.000,C 90.000,E1 305.471} C_DIS
LIN {X -0.230,Y -631.976,Z 568.493,A 0.000,B 0.000,C 90.000,E1 304.739} C_DIS
LIN {X 0.153,Y -636.986,Z 568.489,A 0.000,B 0.000,C 90.000,E1 304.072} C_DIS
LIN {X -0.082,Y -643.482,Z 568.485,A 0.000,B 0.000,C 90.000,E1 303.214} C_DIS
LIN {X 0.031,Y -646.797,Z 568.482,A 0.000,B 0.000,C 90.000,E1 302.704} C_DIS
LIN {X 0.013,Y -650.475,Z 568.478,A 0.000,B 0.000,C 90.000,E1 302.084} C_DIS
LIN {X -0.112,Y -651.731,Z 568.477,A 0.000,B 0.000,C 90.000,E1 301.848} C_DIS
LIN {X 0.193,Y -653.071,Z 568.476,A 0.000,B 0.000,C 90.000,E1 301.592} C_DIS
LIN {X -0.075,Y -656.502,Z 568.472,A 0.000,B 0.000,C 90.000,E1 300.875} C_DIS
LIN {X 0.151,Y -660.789,Z 568.466,A 0.000,B 0.000,C 90.000,E1 299.873} C_DIS
LIN {X -0.033,Y -663.735,Z 568.462,A 0.000,B 0.000,C 90.000,E1 299.155} C_DIS
LIN {X -0.037,Y -667.311,Z 568.457,A 0.000,B 0.000,C 90.000,E1 298.180} C_DIS
LIN {X 0.172,Y -671.552,Z 568.450,A 0.000,B 0.000,C 90.000,E1 296.950} C_DIS
LIN {X -0.088,Y -673.026,Z 568.447,A 0.000,B 0.000,C 90.000,E1 296.488} C_DIS
LIN {X 0.087,Y -673.636,Z 568.446,A 0.000,B 0.000,C 90.000,E1 296.232} C_DIS
LIN {X -0.166,Y -674.302,Z 568.443,A 0.000,B 0.000,C 90.000,E1 295.771} C_DIS
LIN {X -0.278,Y -674.219,Z 568.442,A 0.000,B 0.000,C 90.000,E1 295.540} C_DIS
LIN {X 0.083,Y -672.415,Z 568.439,A 0.000,B 0.000,C 90.000,E1 295.027} C_DIS
LIN {X 0.258,Y -671.004,Z 568.438,A 0.000,B 0.000,C 90.000,E1 294.771} C_DIS
LIN {X 0.172,Y -665.772,Z 568.435,A 0.000,B 0.000,C 90.000,E1 294.259} C_DIS
LIN {X 0.002,Y -663.968,Z 568.434,A 0.000,B 0.000,C 90.000,E1 294.155} C_DIS
LIN {X 0.120,Y -659.146,Z 568.433,A 0.000,B 0.000,C 90.000,E1 293.951} C_DIS
LIN {X 0.069,Y -656.575,Z 568.432,A 0.000,B 0.000,C 90.000,E1 293.823} C_DIS
LIN {X -0.154,Y -654.584,Z 568.432,A 0.000,B 0.000,C 90.000,E1 293.770} C_DIS
LIN {X -0.113,Y -651.959,Z 568.432,A 0.000,B 0.000,C 90.000,E1 293.695} C_DIS
LIN {X -0.016,Y -649.002,Z 568.431,A 0.000,B 0.000,C 90.000,E1 293.590} C_DIS
LIN {X -0.322,Y -645.435,Z 568.431,A 0.000,B 0.000,C 90.000,E1 293.515} C_DIS
LIN {X -0.158,Y -633.935,Z 568.429,A 0.000,B 0.000,C 90.000,E1 293.206} C_DIS
LIN {X 0.323,Y -620.392,Z 568.427,A 0.000,B 0.000,C 90.000,E1 292.823} C_DIS
LIN {X -0.201,Y -599.910,Z 568.424,A 0.000,B 0.000,C 90.000,E1 292.280} C_DIS
LIN {X 0.015,Y -579.360,Z 568.420,A 0.000,B 0.000,C 90.000,E1 291.589} C_DIS
LIN {X 0.054,Y -573.357,Z 568.419,A 0.000,B 0.000,C 90.000,E1 291.354} C_DIS
LIN {X 0.071,Y -568.226,Z 568.417,A 0.000,B 0.000,C 90.000,E1 291.099} C_DIS
LIN {X -0.211,Y -566.974,Z 568.417,A 0.000,B 0.000,C 90.000,E1 291.046} C_DIS
LIN {X 0.024,Y -565.161,Z 568.416,A 0.000,B 0.000,C 90.000,E1 290.865} C_DIS
LIN {X -0.013,Y -565.144,Z 568.416,A 0.000,B 0.000,C 90.000,E1 290.865} C_DIS
LIN {X 0.176,Y -564.529,Z 568.415,A 0.000,B 0.000,C 90.000,E1 290.684} C_DIS
LIN {X 0.077,Y -564.341,Z 568.414,A 0.000,B 0.000,C 90.000,E1 290.556} C_DIS
LIN {X 0.303,Y -564.155,Z 568.412,A 0.000,B 0.000,C 90.000,E1 290.120} C_DIS
LIN {X 0.159,Y -564.189,Z 568.406,A 0.000,B 0.000,C 90.000,E1 289.033} C_DIS
LIN {X 0.018,Y -564.078,Z 568.400,A 0.000,B 0.000,C 90.000,E1 287.946} C_DIS
LIN {X -0.128,Y -563.705,Z 568.394,A 0.000,B 0.000,C 90.000,E1 286.858} C_DIS
LIN {X -0.138,Y -563.061,Z 568.386,A 0.000,B 0.000,C 90.000,E1 285.481} C_DIS
LIN {X 0.231,Y -562.307,Z 568.378,A 0.000,B 0.000,C 90.000,E1 284.064} C_DIS
LIN {X -0.205,Y -561.192,Z 568.368,A 0.000,B 0.000,C 90.000,E1 282.175} C_DIS
LIN {X 0.047,Y -560.186,Z 568.358,A 0.000,B 0.000,C 90.000,E1 280.489} C_DIS
LIN {X 0.143,Y -559.393,Z 568.351,A 0.000,B 0.000,C 90.000,E1 279.095} C_DIS
LIN {X -0.195,Y -558.670,Z 568.341,A 0.000,B 0.000,C 90.000,E1 277.466} C_DIS
LIN {X -0.147,Y -557.977,Z 568.332,A 0.000,B 0.000,C 90.000,E1 275.796} C_DIS
LIN {X -0.041,Y -557.234,Z 568.321,A 0.000,B 0.000,C 90.000,E1 273.841} C_DIS
LIN {X -0.095,Y -556.696,Z 568.312,A 0.000,B 0.000,C 90.000,E1 272.178} C_DIS
LIN {X -0.238,Y -556.135,Z 568.304,A 0.000,B 0.000,C 90.000,E1 270.802} C_DIS
LIN {X 0.075,Y -555.667,Z 568.298,A 0.000,B 0.000,C 90.000,E1 269.656} C_DIS
LIN {X -0.011,Y -554.961,Z 568.289,A 0.000,B 0.000,C 90.000,E1 267.993} C_DIS
LIN {X -0.181,Y -554.294,Z 568.281,A 0.000,B 0.000,C 90.000,E1 266.617} C_DIS
LIN {X -0.266,Y -553.388,Z 568.272,A 0.000,B 0.000,C 90.000,E1 264.951} C_DIS
LIN {X 0.113,Y -552.555,Z 568.264,A 0.000,B 0.000,C 90.000,E1 263.514} C_DIS
LIN {X -0.055,Y -551.754,Z 568.258,A 0.000,B 0.000,C 90.000,E1 262.413} C_DIS
LIN {X -0.225,Y -550.747,Z 568.252,A 0.000,B 0.000,C 90.000,E1 261.310} C_DIS
LIN {X 0.245,Y -549.250,Z 568.244,A 0.000,B 0.000,C 90.000,E1 259.859} C_DIS
LIN {X 0.240,Y -547.522,Z 568.234,A 0.000,B 0.000,C 90.000,E1 258.173} C_DIS
LIN {X -0.114,Y -545.754,Z 568.225,A 0.000,B 0.000,C 90.000,E1 256.520} C_DIS
LIN {X 0.032,Y -543.895,Z 568.216,A 0.000,B 0.000,C 90.000,E1 254.810} C_DIS
LIN {X 0.195,Y -542.126,Z 568.208,A 0.000,B 0.000,C 90.000,E1 253.378} C_DIS
LIN {X -0.192,Y -540.157,Z 568.200,A 0.000,B 0.000,C 90.000,E1 252.000} C_DIS
LIN {X 0.061,Y -537.945,Z 568.192,A 0.000,B 0.000,C 90.000,E1 250.550} C_DIS
LIN {X -0.050,Y -535.516,Z 568.184,A 0.000,B 0.000,C 90.000,E1 249.135} C_DIS
LIN {X -0.199,Y -532.711,Z 568.176,A 0.000,B 0.000,C 90.000,E1 247.720} C_DIS
LIN {X 0.101,Y -530.313,Z 568.170,A 0.000,B 0.000,C 90.000,E1 246.538} C_DIS
LIN {X -0.122,Y -527.831,Z 568.163,A 0.000,B 0.000,C 90.000,E1 245.409} C_DIS
LIN {X 0.009,Y -524.541,Z 568.155,A 0.000,B 0.000,C 90.000,E1 243.948} C_DIS
LIN {X 0.074,Y -521.066,Z 568.147,A 0.000,B 0.000,C 90.000,E1 242.487} C_DIS
LIN {X 0.180,Y -518.135,Z 568.141,A 0.000,B 0.000,C 90.000,E1 241.307} C_DIS
LIN {X -0.119,Y -515.890,Z 568.136,A 0.000,B 0.000,C 90.000,E1 240.461} C_DIS
LIN {X 0.258,Y -513.446,Z 568.131,A 0.000,B 0.000,C 90.000,E1 239.537} C_DIS
LIN {X -0.054,Y -507.369,Z 568.119,A 0.000,B 0.000,C 90.000,E1 237.502} C_DIS
LIN {X -0.006,Y -503.116,Z 568.111,A 0.000,B 0.000,C 90.000,E1 236.008} C_DIS
LIN {X 0.234,Y -498.866,Z 568.103,A 0.000,B 0.000,C 90.000,E1 234.482} C_DIS
LIN {X 0.001,Y -493.125,Z 568.091,A 0.000,B 0.000,C 90.000,E1 232.396} C_DIS
LIN {X 0.099,Y -489.848,Z 568.084,A 0.000,B 0.000,C 90.000,E1 231.170} C_DIS
LIN {X -0.093,Y -485.920,Z 568.076,A 0.000,B 0.000,C 90.000,E1 229.666} C_DIS
LIN {X 0.133,Y -481.254,Z 568.066,A 0.000,B 0.000,C 90.000,E1 227.796} C_DIS
LIN {X 0.079,Y -475.070,Z 568.052,A 0.000,B 0.000,C 90.000,E1 225.324} C_DIS
LIN {X 0.001,Y -470.643,Z 568.042,A 0.000,B 0.000,C 90.000,E1 223.461} C_DIS
LIN {X -0.231,Y -467.028,Z 568.033,A 0.000,B 0.000,C 90.000,E1 221.919} C_DIS
LIN {X -0.126,Y -462.746,Z 568.022,A 0.000,B 0.000,C 90.000,E1 220.011} C_DIS
LIN {X -0.194,Y -460.042,Z 568.015,A 0.000,B 0.000,C 90.000,E1 218.749} C_DIS
LIN {X 0.160,Y -455.901,Z 568.005,A 0.000,B 0.000,C 90.000,E1 216.790} C_DIS
LIN {X -0.210,Y -452.556,Z 567.996,A 0.000,B 0.000,C 90.000,E1 215.231} C_DIS
LIN {X -0.196,Y -448.660,Z 567.985,A 0.000,B 0.000,C 90.000,E1 213.293} C_DIS
LIN {X -0.138,Y -444.879,Z 567.974,A 0.000,B 0.000,C 90.000,E1 211.337} C_DIS
LIN {X 0.158,Y -441.917,Z 567.965,A 0.000,B 0.000,C 90.000,E1 209.667} C_DIS
LIN {X 0.034,Y -437.890,Z 567.952,A 0.000,B 0.000,C 90.000,E1 207.385} C_DIS
LIN {X -0.024,Y -434.485,Z 567.941,A 0.000,B 0.000,C 90.000,E1 205.412} C_DIS
LIN {X 0.045,Y -430.651,Z 567.928,A 0.000,B 0.000,C 90.000,E1 203.078} C_DIS
LIN {X -0.133,Y -426.603,Z 567.913,A 0.000,B 0.000,C 90.000,E1 200.429} C_DIS
LIN {X -0.144,Y -424.725,Z 567.906,A 0.000,B 0.000,C 90.000,E1 199.087} C_DIS
LIN {X 0.046,Y -421.971,Z 567.895,A 0.000,B 0.000,C 90.000,E1 197.040} C_DIS
LIN {X 0.045,Y -419.442,Z 567.883,A 0.000,B 0.000,C 90.000,E1 195.009} C_DIS
LIN {X 0.069,Y -417.778,Z 567.876,A 0.000,B 0.000,C 90.000,E1 193.647} C_DIS
LIN {X -0.081,Y -416.341,Z 567.870,A 0.000,B 0.000,C 90.000,E1 192.647} C_DIS
LIN {X -0.031,Y -412.592,Z 567.855,A 0.000,B 0.000,C 90.000,E1 189.905} C_DIS
LIN {X 0.179,Y -410.118,Z 567.844,A 0.000,B 0.000,C 90.000,E1 187.814} C_DIS
LIN {X -0.207,Y -408.293,Z 567.834,A 0.000,B 0.000,C 90.000,E1 186.144} C_DIS
LIN {X 0.187,Y -406.460,Z 567.824,A 0.000,B 0.000,C 90.000,E1 184.359} C_DIS
LIN {X -0.068,Y -402.999,Z 567.803,A 0.000,B 0.000,C 90.000,E1 180.573} C_DIS
LIN {X 0.115,Y -401.558,Z 567.792,A 0.000,B 0.000,C 90.000,E1 178.453} C_DIS
LIN {X -0.067,Y -400.587,Z 567.782,A 0.000,B 0.000,C 90.000,E1 176.731} C_DIS
LIN {X 0.043,Y -399.559,Z 567.766,A 0.000,B 0.000,C 90.000,E1 173.913} C_DIS
LIN {X -0.175,Y -399.137,Z 567.753,A 0.000,B 0.000,C 90.000,E1 171.489} C_DIS
LIN {X 0.097,Y -399.019,Z 567.739,A 0.000,B 0.000,C 90.000,E1 168.993} C_DIS
LIN {X -0.222,Y -399.378,Z 567.721,A 0.000,B 0.000,C 90.000,E1 165.880} C_DIS
LIN {X -0.019,Y -399.764,Z 567.714,A 0.000,B 0.000,C 90.000,E1 164.448} C_DIS
LIN {X 0.033,Y -400.653,Z 567.698,A 0.000,B 0.000,C 90.000,E1 161.638} C_DIS
LIN {X 0.176,Y -401.606,Z 567.686,A 0.000,B 0.000,C 90.000,E1 159.518} C_DIS
LIN {X 0.097,Y -402.616,Z 567.675,A 0.000,B 0.000,C 90.000,E1 157.433} C_DIS
LIN {X -0.019,Y -403.773,Z 567.663,A 0.000,B 0.000,C 90.000,E1 155.357} C_DIS
LIN {X 0.072,Y -404.924,Z 567.652,A 0.000,B 0.000,C 90.000,E1 153.256} C_DIS
LIN {X 0.110,Y -405.921,Z 567.642,A 0.000,B 0.000,C 90.000,E1 151.513} C_DIS
LIN {X 0.095,Y -406.609,Z 567.634,A 0.000,B 0.000,C 90.000,E1 150.127} C_DIS
LIN {X 0.091,Y -407.228,Z 567.626,A 0.000,B 0.000,C 90.000,E1 148.742} C_DIS
LIN {X -0.126,Y -407.869,Z 567.617,A 0.000,B 0.000,C 90.000,E1 147.041} C_DIS
LIN {X -0.103,Y -408.295,Z 567.607,A 0.000,B 0.000,C 90.000,E1 145.308} C_DIS
LIN {X -0.077,Y -408.637,Z 567.598,A 0.000,B 0.000,C 90.000,E1 143.577} C_DIS
LIN {X 0.109,Y -408.933,Z 567.588,A 0.000,B 0.000,C 90.000,E1 141.823} C_DIS
LIN {X 0.151,Y -409.094,Z 567.580,A 0.000,B 0.000,C 90.000,E1 140.436} C_DIS
LIN {X 0.027,Y -409.249,Z 567.571,A 0.000,B 0.000,C 90.000,E1 138.728} C_DIS
LIN {X -0.009,Y -409.338,Z 567.559,A 0.000,B 0.000,C 90.000,E1 136.662} C_DIS
LIN {X -0.180,Y -409.588,Z 567.546,A 0.000,B 0.000,C 90.000,E1 134.271} C_DIS
LIN {X -0.050,Y -409.837,Z 567.536,A 0.000,B 0.000,C 90.000,E1 132.528} C_DIS
LIN {X -0.045,Y -409.932,Z 567.529,A 0.000,B 0.000,C 90.000,E1 131.148} C_DIS
LIN {X -0.044,Y -409.837,Z 567.521,A 0.000,B 0.000,C 90.000,E1 129.769} C_DIS
LIN {X -0.149,Y -409.694,Z 567.515,A 0.000,B 0.000,C 90.000,E1 128.749} C_DIS
LIN {X -0.143,Y -409.574,Z 567.511,A 0.000,B 0.000,C 90.000,E1 128.016} C_DIS
LIN {X 0.075,Y -415.522,Z 567.500,A 0.000,B 0.000,C 90.000,E1 125.964} C_DIS
LIN {X 0.159,Y -425.914,Z 567.477,A 0.000,B 0.000,C 90.000,E1 121.878} C_DIS
LIN {X 0.113,Y -430.927,Z 567.468,A 0.000,B 0.000,C 90.000,E1 120.207} C_DIS
LIN {X -0.141,Y -436.293,Z 567.455,A 0.000,B 0.000,C 90.000,E1 117.975} C_DIS
LIN {X -0.181,Y -436.358,Z 567.455,A 0.000,B 0.000,C 90.000,E1 117.975} C_DIS
LIN {X -0.052,Y -444.381,Z 567.453,A 0.000,B 0.000,C 90.000,E1 117.590} C_DIS
LIN {X 0.123,Y -463.565,Z 567.448,A 0.000,B 0.000,C 90.000,E1 116.693} C_DIS
LIN {X 0.039,Y -480.708,Z 567.444,A 0.000,B 0.000,C 90.000,E1 115.899} C_DIS
LIN {X -0.124,Y -489.062,Z 567.442,A 0.000,B 0.000,C 90.000,E1 115.515} C_DIS
LIN {X 0.118,Y -499.063,Z 567.439,A 0.000,B 0.000,C 90.000,E1 114.975} C_DIS
LIN {X 0.203,Y -510.576,Z 567.435,A 0.000,B 0.000,C 90.000,E1 114.335} C_DIS
LIN {X -0.116,Y -517.047,Z 567.433,A 0.000,B 0.000,C 90.000,E1 114.003} C_DIS
LIN {X 0.291,Y -526.684,Z 567.430,A 0.000,B 0.000,C 90.000,E1 113.387} C_DIS
LIN {X -0.069,Y -537.567,Z 567.426,A 0.000,B 0.000,C 90.000,E1 112.717} C_DIS
LIN {X -0.190,Y -547.986,Z 567.422,A 0.000,B 0.000,C 90.000,E1 111.972} C_DIS
LIN {X 0.225,Y -553.693,Z 567.419,A 0.000,B 0.000,C 90.000,E1 111.461} C_DIS
LIN {X 0.257,Y -559.203,Z 567.417,A 0.000,B 0.000,C 90.000,E1 110.972} C_DIS
LIN {X 0.166,Y -565.139,Z 567.413,A 0.000,B 0.000,C 90.000,E1 110.375} C_DIS
LIN {X -0.182,Y -569.858,Z 567.410,A 0.000,B 0.000,C 90.000,E1 109.866} C_DIS
LIN {X -0.125,Y -573.052,Z 567.408,A 0.000,B 0.000,C 90.000,E1 109.450} C_DIS
LIN {X 0.230,Y -574.981,Z 567.406,A 0.000,B 0.000,C 90.000,E1 109.141} C_DIS
LIN {X 0.233,Y -578.706,Z 567.404,A 0.000,B 0.000,C 90.000,E1 108.598} C_DIS
LIN {X -0.082,Y -583.653,Z 567.399,A 0.000,B 0.000,C 90.000,E1 107.819} C_DIS
LIN {X -0.098,Y -587.431,Z 567.395,A 0.000,B 0.000,C 90.000,E1 107.149} C_DIS
LIN {X -0.185,Y -591.559,Z 567.391,A 0.000,B 0.000,C 90.000,E1 106.370} C_DIS
LIN {X 0.143,Y -596.003,Z 567.386,A 0.000,B 0.000,C 90.000,E1 105.426} C_DIS
LIN {X -0.156,Y -600.186,Z 567.381,A 0.000,B 0.000,C 90.000,E1 104.537} C_DIS
LIN {X 0.348,Y -605.734,Z 567.373,A 0.000,B 0.000,C 90.000,E1 103.175} C_DIS
LIN {X 0.091,Y -611.019,Z 567.366,A 0.000,B 0.000,C 90.000,E1 101.895} C_DIS
LIN {X 0.049,Y -616.018,Z 567.359,A 0.000,B 0.000,C 90.000,E1 100.602} C_DIS
LIN {X 0.020,Y -622.747,Z 567.349,A 0.000,B 0.000,C 90.000,E1 98.803} C_DIS
LIN {X -0.041,Y -627.419,Z 567.342,A 0.000,B 0.000,C 90.000,E1 97.530} C_DIS
LIN {X 0.258,Y -630.983,Z 567.336,A 0.000,B 0.000,C 90.000,E1 96.486} C_DIS
LIN {X 0.109,Y -633.471,Z 567.332,A 0.000,B 0.000,C 90.000,E1 95.739} C_DIS
LIN {X -0.012,Y -635.774,Z 567.328,A 0.000,B 0.000,C 90.000,E1 94.992} C_DIS
LIN {X 0.319,Y -638.488,Z 567.322,A 0.000,B 0.000,C 90.000,E1 93.955} C_DIS
LIN {X -0.001,Y -640.904,Z 567.317,A 0.000,B 0.000,C 90.000,E1 92.980} C_DIS
LIN {X -0.318,Y -642.780,Z 567.311,A 0.000,B 0.000,C 90.000,E1 92.007} C_DIS
LIN {X 0.287,Y -643.949,Z 567.307,A 0.000,B 0.000,C 90.000,E1 91.203} C_DIS
LIN {X 0.244,Y -644.864,Z 567.303,A 0.000,B 0.000,C 90.000,E1 90.458} C_DIS
LIN {X 0.212,Y -645.536,Z 567.299,A 0.000,B 0.000,C 90.000,E1 89.714} C_DIS
LIN {X 0.185,Y -645.871,Z 567.294,A 0.000,B 0.000,C 90.000,E1 88.969} C_DIS
LIN {X -0.046,Y -645.868,Z 567.289,A 0.000,B 0.000,C 90.000,E1 87.993} C_DIS
LIN {X -0.075,Y -645.586,Z 567.285,A 0.000,B 0.000,C 90.000,E1 87.249} C_DIS
LIN {X -0.308,Y -644.857,Z 567.279,A 0.000,B 0.000,C 90.000,E1 86.274} C_DIS
LIN {X 0.090,Y -643.678,Z 567.274,A 0.000,B 0.000,C 90.000,E1 85.241} C_DIS
LIN {X 0.127,Y -642.712,Z 567.269,A 0.000,B 0.000,C 90.000,E1 84.489} C_DIS
LIN {X -0.155,Y -640.996,Z 567.264,A 0.000,B 0.000,C 90.000,E1 83.514} C_DIS
LIN {X 0.323,Y -638.876,Z 567.258,A 0.000,B 0.000,C 90.000,E1 82.470} C_DIS
LIN {X -0.121,Y -637.704,Z 567.256,A 0.000,B 0.000,C 90.000,E1 82.008} C_DIS
LIN {X 0.224,Y -635.140,Z 567.250,A 0.000,B 0.000,C 90.000,E1 80.971} C_DIS
LIN {X -0.189,Y -631.505,Z 567.243,A 0.000,B 0.000,C 90.000,E1 79.746} C_DIS
LIN {X 0.159,Y -628.342,Z 567.237,A 0.000,B 0.000,C 90.000,E1 78.701} C_DIS
LIN {X 0.174,Y -625.834,Z 567.233,A 0.000,B 0.000,C 90.000,E1 77.937} C_DIS
LIN {X 0.168,Y -623.063,Z 567.229,A 0.000,B 0.000,C 90.000,E1 77.173} C_DIS
LIN {X -0.254,Y -621.103,Z 567.226,A 0.000,B 0.000,C 90.000,E1 76.700} C_DIS
LIN {X -0.305,Y -617.840,Z 567.222,A 0.000,B 0.000,C 90.000,E1 75.936} C_DIS
LIN {X 0.202,Y -614.376,Z 567.217,A 0.000,B 0.000,C 90.000,E1 75.117} C_DIS
LIN {X -0.316,Y -611.335,Z 567.214,A 0.000,B 0.000,C 90.000,E1 74.519} C_DIS
LIN {X -0.314,Y -607.351,Z 567.210,A 0.000,B 0.000,C 90.000,E1 73.740} C_DIS
LIN {X -0.303,Y -603.733,Z 567.206,A 0.000,B 0.000,C 90.000,E1 73.087} C_DIS
LIN {X -0.018,Y -600.825,Z 567.203,A 0.000,B 0.000,C 90.000,E1 72.543} C_DIS
LIN {X 0.116,Y -596.817,Z 567.199,A 0.000,B 0.000,C 90.000,E1 71.873} C_DIS
LIN {X 0.226,Y -591.456,Z 567.195,A 0.000,B 0.000,C 90.000,E1 71.094} C_DIS
LIN {X -0.211,Y -587.560,Z 567.192,A 0.000,B 0.000,C 90.000,E1 70.604} C_DIS
LIN {X -0.050,Y -584.206,Z 567.190,A 0.000,B 0.000,C 90.000,E1 70.188} C_DIS
LIN {X -0.187,Y -582.038,Z 567.188,A 0.000,B 0.000,C 90.000,E1 69.934} C_DIS
LIN {X -0.136,Y -577.314,Z 567.185,A 0.000,B 0.000,C 90.000,E1 69.390} C_DIS
LIN {X -0.068,Y -572.160,Z 567.182,A 0.000,B 0.000,C 90.000,E1 68.847} C_DIS
LIN {X -0.175,Y -568.201,Z 567.180,A 0.000,B 0.000,C 90.000,E1 68.465} C_DIS
LIN {X 0.204,Y -562.643,Z 567.177,A 0.000,B 0.000,C 90.000,E1 67.922} C_DIS
LIN {X -0.171,Y -556.775,Z 567.175,A 0.000,B 0.000,C 90.000,E1 67.486} C_DIS
LIN {X -0.232,Y -550.607,Z 567.172,A 0.000,B 0.000,C 90.000,E1 67.050} C_DIS
LIN {X -0.247,Y -545.772,Z 567.171,A 0.000,B 0.000,C 90.000,E1 66.741} C_DIS
LIN {X 0.173,Y -539.009,Z 567.169,A 0.000,B 0.000,C 90.000,E1 66.305} C_DIS
LIN {X -0.021,Y -532.131,Z 567.167,A 0.000,B 0.000,C 90.000,E1 65.973} C_DIS
LIN {X 0.132,Y -528.818,Z 567.166,A 0.000,B 0.000,C 90.000,E1 65.793} C_DIS
LIN {X -0.055,Y -516.491,Z 567.163,A 0.000,B 0.000,C 90.000,E1 65.281} C_DIS
LIN {X 0.157,Y -509.376,Z 567.161,A 0.000,B 0.000,C 90.000,E1 64.973} C_DIS
LIN {X -0.111,Y -484.764,Z 567.156,A 0.000,B 0.000,C 90.000,E1 64.076} C_DIS
LIN {X -0.067,Y -462.513,Z 567.151,A 0.000,B 0.000,C 90.000,E1 63.179} C_DIS
LIN {X 0.039,Y -457.242,Z 567.150,A 0.000,B 0.000,C 90.000,E1 62.922} C_DIS
LIN {X 0.000,Y -457.167,Z 567.150,A 0.000,B 0.000,C 90.000,E1 62.922} C_DIS
LIN {X 0.119,Y -455.499,Z 567.144,A 0.000,B 0.000,C 90.000,E1 61.897} C_DIS
LIN {X 0.124,Y -445.550,Z 567.119,A 0.000,B 0.000,C 90.000,E1 57.375} C_DIS
LIN {X -0.059,Y -443.761,Z 567.113,A 0.000,B 0.000,C 90.000,E1 56.421} C_DIS
LIN {X 0.057,Y -437.971,Z 567.100,A 0.000,B 0.000,C 90.000,E1 54.036} C_DIS
LIN {X 0.018,Y -437.973,Z 567.100,A 0.000,B 0.000,C 90.000,E1 54.036} C_DIS
LIN {X -0.056,Y -440.689,Z 567.088,A 0.000,B 0.000,C 90.000,E1 51.823} C_DIS
LIN {X 0.216,Y -441.923,Z 567.082,A 0.000,B 0.000,C 90.000,E1 50.803} C_DIS
LIN {X 0.119,Y -444.304,Z 567.072,A 0.000,B 0.000,C 90.000,E1 48.852} C_DIS
LIN {X 0.054,Y -446.212,Z 567.063,A 0.000,B 0.000,C 90.000,E1 47.229} C_DIS
LIN {X -0.297,Y -447.697,Z 567.055,A 0.000,B 0.000,C 90.000,E1 45.972} C_DIS
LIN {X 0.005,Y -448.714,Z 567.050,A 0.000,B 0.000,C 90.000,E1 44.960} C_DIS
LIN {X -0.314,Y -449.568,Z 567.044,A 0.000,B 0.000,C 90.000,E1 44.028} C_DIS
LIN {X 0.017,Y -450.329,Z 567.039,A 0.000,B 0.000,C 90.000,E1 43.014} C_DIS
LIN {X -0.273,Y -451.118,Z 567.032,A 0.000,B 0.000,C 90.000,E1 41.757} C_DIS
LIN {X -0.220,Y -451.675,Z 567.025,A 0.000,B 0.000,C 90.000,E1 40.458} C_DIS
LIN {X 0.185,Y -451.938,Z 567.018,A 0.000,B 0.000,C 90.000,E1 39.116} C_DIS
LIN {X -0.046,Y -452.077,Z 567.010,A 0.000,B 0.000,C 90.000,E1 37.855} C_DIS
LIN {X 0.152,Y -451.935,Z 567.001,A 0.000,B 0.000,C 90.000,E1 36.217} C_DIS
LIN {X 0.030,Y -451.753,Z 566.996,A 0.000,B 0.000,C 90.000,E1 35.264} C_DIS
LIN {X 0.010,Y -451.115,Z 566.983,A 0.000,B 0.000,C 90.000,E1 33.007} C_DIS
LIN {X 0.139,Y -450.684,Z 566.973,A 0.000,B 0.000,C 90.000,E1 31.052} C_DIS
LIN {X -0.058,Y -450.444,Z 566.964,A 0.000,B 0.000,C 90.000,E1 29.461} C_DIS
LIN {X -0.002,Y -450.049,Z 566.953,A 0.000,B 0.000,C 90.000,E1 27.513} C_DIS
LIN {X -0.160,Y -449.631,Z 566.942,A 0.000,B 0.000,C 90.000,E1 25.591} C_DIS
LIN {X 0.133,Y -449.495,Z 566.935,A 0.000,B 0.000,C 90.000,E1 24.259} C_DIS
LIN {X 0.171,Y -449.295,Z 566.921,A 0.000,B 0.000,C 90.000,E1 21.663} C_DIS
LIN {X 0.168,Y -449.232,Z 566.908,A 0.000,B 0.000,C 90.000,E1 19.396} C_DIS
LIN {X 0.130,Y -449.336,Z 566.897,A 0.000,B 0.000,C 90.000,E1 17.457} C_DIS
LIN {X -0.126,Y -449.732,Z 566.883,A 0.000,B 0.000,C 90.000,E1 14.898} C_DIS
LIN {X 0.010,Y -450.278,Z 566.872,A 0.000,B 0.000,C 90.000,E1 12.939} C_DIS
LIN {X 0.145,Y -451.184,Z 566.859,A 0.000,B 0.000,C 90.000,E1 10.658} C_DIS
LIN {X 0.152,Y -452.377,Z 566.847,A 0.000,B 0.000,C 90.000,E1 8.398} C_DIS
LIN {X 0.053,Y -454.282,Z 566.831,A 0.000,B 0.000,C 90.000,E1 5.511} C_DIS
LIN {X -0.177,Y -455.845,Z 566.820,A 0.000,B 0.000,C 90.000,E1 3.612} C_DIS
LIN {X -0.035,Y -458.233,Z 566.806,A 0.000,B 0.000,C 90.000,E1 1.031} C_DIS
LIN {X -0.149,Y -460.667,Z 566.794,A 0.000,B 0.000,C 90.000,E1 358.854} C_DIS
LIN {X -0.056,Y -463.572,Z 566.781,A 0.000,B 0.000,C 90.000,E1 356.617} C_DIS
LIN {X 0.151,Y -466.673,Z 566.769,A 0.000,B 0.000,C 90.000,E1 354.375} C_DIS
LIN {X -0.010,Y -469.034,Z 566.760,A 0.000,B 0.000,C 90.000,E1 352.818} C_DIS
LIN {X -0.065,Y -471.339,Z 566.751,A 0.000,B 0.000,C 90.000,E1 351.254} C_DIS
LIN {X 0.047,Y -474.599,Z 566.739,A 0.000,B 0.000,C 90.000,E1 349.050} C_DIS
LIN {X -0.198,Y -476.990,Z 566.731,A 0.000,B 0.000,C 90.000,E1 347.521} C_DIS
LIN {X -0.110,Y -480.511,Z 566.719,A 0.000,B 0.000,C 90.000,E1 345.338} C_DIS
LIN {X 0.049,Y -485.583,Z 566.703,A 0.000,B 0.000,C 90.000,E1 342.543} C_DIS
LIN {X -0.182,Y -489.113,Z 566.693,A 0.000,B 0.000,C 90.000,E1 340.732} C_DIS
LIN {X -0.208,Y -492.093,Z 566.684,A 0.000,B 0.000,C 90.000,E1 339.209} C_DIS
LIN {X -0.049,Y -494.327,Z 566.678,A 0.000,B 0.000,C 90.000,E1 337.975} C_DIS
LIN {X -0.259,Y -497.207,Z 566.669,A 0.000,B 0.000,C 90.000,E1 336.485} C_DIS
LIN {X -0.217,Y -499.901,Z 566.661,A 0.000,B 0.000,C 90.000,E1 334.973} C_DIS
LIN {X 0.163,Y -502.951,Z 566.651,A 0.000,B 0.000,C 90.000,E1 333.127} C_DIS
LIN {X -0.226,Y -504.895,Z 566.644,A 0.000,B 0.000,C 90.000,E1 331.975} C_DIS
LIN {X -0.032,Y -507.348,Z 566.636,A 0.000,B 0.000,C 90.000,E1 330.461} C_DIS
LIN {X 0.074,Y -511.315,Z 566.623,A 0.000,B 0.000,C 90.000,E1 328.074} C_DIS
LIN {X 0.131,Y -514.340,Z 566.613,A 0.000,B 0.000,C 90.000,E1 326.294} C_DIS
LIN {X -0.106,Y -516.911,Z 566.605,A 0.000,B 0.000,C 90.000,E1 324.848} C_DIS
LIN {X -0.003,Y -519.524,Z 566.597,A 0.000,B 0.000,C 90.000,E1 323.371} C_DIS
LIN {X -0.095,Y -523.769,Z 566.584,A 0.000,B 0.000,C 90.000,E1 321.045} C_DIS
LIN {X 0.213,Y -528.473,Z 566.571,A 0.000,B 0.000,C 90.000,E1 318.690} C_DIS
LIN {X -0.037,Y -532.404,Z 566.561,A 0.000,B 0.000,C 90.000,E1 316.986} C_DIS
LIN {X -0.240,Y -537.193,Z 566.550,A 0.000,B 0.000,C 90.000,E1 315.000} C_DIS
LIN {X -0.308,Y -540.242,Z 566.544,A 0.000,B 0.000,C 90.000,E1 313.866} C_DIS
LIN {X 0.067,Y -542.008,Z 566.540,A 0.000,B 0.000,C 90.000,E1 313.257} C_DIS
LIN {X 0.049,Y -543.083,Z 566.539,A 0.000,B 0.000,C 90.000,E1 312.975} C_DIS
LIN {X -0.035,Y -544.357,Z 566.538,A 0.000,B 0.000,C 90.000,E1 312.771} C_DIS
LIN {X 0.000,Y -546.215,Z 566.535,A 0.000,B 0.000,C 90.000,E1 312.366} C_DIS
LIN {X 0.026,Y -548.219,Z 566.534,A 0.000,B 0.000,C 90.000,E1 312.081} C_DIS
LIN {X -0.346,Y -550.143,Z 566.532,A 0.000,B 0.000,C 90.000,E1 311.838} C_DIS
LIN {X 0.063,Y -552.360,Z 566.531,A 0.000,B 0.000,C 90.000,E1 311.515} C_DIS
LIN {X 0.318,Y -556.573,Z 566.528,A 0.000,B 0.000,C 90.000,E1 311.067} C_DIS
LIN {X 0.232,Y -560.855,Z 566.526,A 0.000,B 0.000,C 90.000,E1 310.701} C_DIS
LIN {X -0.273,Y -569.347,Z 566.523,A 0.000,B 0.000,C 90.000,E1 310.092} C_DIS
LIN {X -0.086,Y -576.640,Z 566.520,A 0.000,B 0.000,C 90.000,E1 309.564} C_DIS
LIN {X 0.049,Y -589.908,Z 566.514,A 0.000,B 0.000,C 90.000,E1 308.588} C_DIS
LIN {X -0.225,Y -595.445,Z 566.512,A 0.000,B 0.000,C 90.000,E1 308.177} C_DIS
LIN {X 0.119,Y -600.811,Z 566.509,A 0.000,B 0.000,C 90.000,E1 307.684} C_DIS
LIN {X -0.250,Y -606.012,Z 566.507,A 0.000,B 0.000,C 90.000,E1 307.237} C_DIS
LIN {X -0.282,Y -609.811,Z 566.505,A 0.000,B 0.000,C 90.000,E1 306.870} C_DIS
LIN {X -0.044,Y -614.625,Z 566.502,A 0.000,B 0.000,C 90.000,E1 306.343} C_DIS
LIN {X -0.342,Y -621.555,Z 566.498,A 0.000,B 0.000,C 90.000,E1 305.598} C_DIS
LIN {X -0.227,Y -629.130,Z 566.493,A 0.000,B 0.000,C 90.000,E1 304.692} C_DIS
LIN {X -0.029,Y -635.274,Z 566.488,A 0.000,B 0.000,C 90.000,E1 303.913} C_DIS
LIN {X -0.159,Y -639.148,Z 566.486,A 0.000,B 0.000,C 90.000,E1 303.420} C_DIS
LIN {X -0.102,Y -641.946,Z 566.484,A 0.000,B 0.000,C 90.000,E1 303.038} C_DIS
LIN {X -0.220,Y -644.611,Z 566.481,A 0.000,B 0.000,C 90.000,E1 302.673} C_DIS
LIN {X -0.227,Y -649.068,Z 566.477,A 0.000,B 0.000,C 90.000,E1 301.926} C_DIS
LIN {X -0.064,Y -651.762,Z 566.475,A 0.000,B 0.000,C 90.000,E1 301.416} C_DIS
LIN {X 0.002,Y -655.268,Z 566.470,A 0.000,B 0.000,C 90.000,E1 300.669} C_DIS
END
